C07285=1043.787,311.118,385.391,172.204,41.135,157.884
C07286=1043.780,310.870,385.424,172.200,41.132,157.883
C07287=1043.773,310.622,385.458,172.196,41.130,157.882
C07288=1043.766,310.375,385.491,172.192,41.127,157.881
C07289=1043.759,310.127,385.525,172.189,41.125,157.880
C07290=1043.751,309.879,385.558,172.185,41.122,157.880
C07291=1043.745,309.632,385.591,172.181,41.119,157.879
C07292=1043.738,309.385,385.625,172.177,41.116,157.878
C07293=1043.731,309.136,385.658,172.173,41.113,157.877
C07294=1043.724,308.889,385.691,172.169,41.111,157.876
C07295=1043.717,308.642,385.725,172.165,41.108,157.875
C07296=1043.710,308.393,385.758,172.161,41.106,157.875
C07297=1043.703,308.146,385.792,172.157,41.103,157.874
C07298=1043.696,307.898,385.824,172.153,41.100,157.873
C07299=1043.689,307.651,385.858,172.149,41.098,157.872
C07300=1043.682,307.404,385.892,172.146,41.095,157.872
C07301=1043.675,307.155,385.925,172.142,41.093,157.871
C07302=1043.669,306.908,385.958,172.138,41.090,157.870
C07303=1043.662,306.660,385.991,172.134,41.087,157.869
C07304=1043.654,306.412,386.025,172.130,41.085,157.868
C07305=1043.647,306.165,386.057,172.126,41.082,157.868
C07306=1043.640,305.918,386.091,172.122,41.079,157.867
C07307=1043.632,305.593,386.135,172.117,41.076,157.866
C07308=1043.623,305.268,386.178,172.112,41.073,157.865
C07309=1043.614,304.942,386.222,172.107,41.070,157.864
C07310=1043.605,304.618,386.265,172.102,41.066,157.863
C07311=1043.597,304.370,386.298,172.099,41.063,157.862
C07312=1043.591,304.123,386.331,172.095,41.060,157.861
C07313=1043.584,303.875,386.364,172.091,41.058,157.860
C07314=1043.578,303.627,386.397,172.087,41.056,157.860
C07315=1043.570,303.379,386.431,172.084,41.053,157.859
C07316=1043.564,303.132,386.464,172.080,41.051,157.858
C07317=1043.557,302.885,386.496,172.076,41.048,157.857
C07318=1043.550,302.636,386.529,172.072,41.045,157.856
C07319=1043.544,302.389,386.563,172.068,41.043,157.856
C07320=1043.537,302.141,386.596,172.065,41.040,157.855
C07321=1043.530,301.893,386.628,172.061,41.037,157.854
C07322=1043.523,301.645,386.661,172.057,41.035,157.853
C07323=1043.516,301.398,386.694,172.054,41.032,157.853
C07324=1043.510,301.151,386.727,172.050,41.030,157.852
C07325=1043.503,300.903,386.760,172.046,41.027,157.851
C07326=1043.497,300.655,386.793,172.042,41.025,157.850
C07327=1043.490,300.407,386.826,172.039,41.022,157.850
C07328=1043.483,300.159,386.858,172.035,41.019,157.849
C07329=1043.476,299.912,386.892,172.031,41.017,157.848
C07330=1043.469,299.664,386.925,172.028,41.015,157.847
C07331=1043.463,299.416,386.957,172.024,41.012,157.847
C07332=1043.457,299.169,386.990,172.020,41.009,157.846
C07333=1043.449,298.921,387.023,172.017,41.007,157.845
C07334=1043.443,298.673,387.055,172.013,41.004,157.844
C07335=1043.436,298.426,387.088,172.009,41.001,157.843
C07336=1043.430,298.178,387.121,172.006,40.999,157.843
C07337=1043.423,297.930,387.153,172.002,40.997,157.842
C07338=1043.416,297.683,387.186,171.999,40.994,157.841
C07339=1043.410,297.435,387.219,171.995,40.991,157.840
C07340=1043.403,297.187,387.252,171.991,40.989,157.840
C07341=1043.397,296.939,387.285,171.988,40.987,157.839
C07342=1043.390,296.692,387.317,171.985,40.984,157.838
C07343=1043.383,296.444,387.350,171.981,40.981,157.837
C07344=1043.377,296.197,387.382,171.977,40.979,157.837
C07345=1043.371,295.948,387.415,171.973,40.976,157.836
C07346=1043.364,295.700,387.447,171.970,40.974,157.835
C07347=1043.357,295.453,387.480,171.967,40.971,157.834
C07348=1043.350,295.206,387.512,171.963,40.969,157.834
C07349=1043.343,294.957,387.545,171.959,40.966,157.833
C07350=1043.337,294.709,387.576,171.956,40.964,157.832
C07351=1043.330,294.462,387.609,171.952,40.962,157.832
C07352=1043.323,294.214,387.641,171.949,40.959,157.831
C07353=1043.317,293.966,387.674,171.945,40.957,157.830
C07354=1043.310,293.718,387.706,171.941,40.954,157.829
C07355=1043.303,293.471,387.739,171.938,40.951,157.829
C07356=1043.297,293.223,387.770,171.934,40.949,157.828
C07357=1043.289,292.975,387.803,171.931,40.947,157.827
C07358=1043.283,292.727,387.835,171.927,40.945,157.827
C07359=1043.276,292.479,387.867,171.924,40.942,157.826
C07360=1043.269,292.232,387.899,171.920,40.940,157.825
C07361=1043.263,291.984,387.931,171.916,40.937,157.824
C07362=1043.255,291.736,387.963,171.914,40.935,157.824
C07363=1043.247,291.427,388.003,171.909,40.932,157.823
C07364=1043.239,291.119,388.043,171.905,40.929,157.822
C07365=1043.231,290.810,388.083,171.900,40.926,157.821
C07366=1043.223,290.502,388.123,171.896,40.923,157.820
C07367=1043.215,290.254,388.154,171.892,40.921,157.820
C07368=1043.208,290.006,388.187,171.889,40.918,157.819
C07369=1043.202,289.758,388.219,171.886,40.916,157.818
C07370=1043.196,289.510,388.250,171.882,40.914,157.817
C07371=1043.188,289.263,388.282,171.879,40.911,157.817
C07372=1043.182,289.015,388.314,171.875,40.909,157.816
C07373=1043.176,288.767,388.346,171.871,40.906,157.815
C07374=1043.169,288.520,388.378,171.869,40.904,157.815
C07375=1043.162,288.272,388.409,171.865,40.902,157.814
C07376=1043.155,288.023,388.441,171.861,40.900,157.813
C07377=1043.148,287.775,388.474,171.859,40.897,157.813
C07378=1043.142,287.528,388.505,171.855,40.895,157.812
C07379=1043.135,287.280,388.537,171.851,40.893,157.811
C07380=1043.128,287.032,388.568,171.848,40.890,157.810
C07381=1043.121,286.785,388.600,171.844,40.888,157.810
C07382=1043.114,286.537,388.632,171.841,40.886,157.809
C07383=1043.108,286.289,388.663,171.838,40.883,157.808
C07384=1043.101,286.041,388.695,171.834,40.881,157.808
C07385=1043.094,285.793,388.726,171.831,40.879,157.807
C07386=1043.088,285.545,388.757,171.828,40.877,157.807
C07387=1043.081,285.297,388.789,171.824,40.874,157.806
C07388=1043.074,285.049,388.820,171.820,40.872,157.805
C07389=1043.067,284.802,388.852,171.818,40.870,157.804
C07390=1043.061,284.554,388.884,171.814,40.867,157.804
C07391=1043.054,284.306,388.916,171.811,40.865,157.803
C07392=1043.048,284.058,388.947,171.807,40.863,157.802
C07393=1043.041,283.810,388.979,171.804,40.861,157.802
C07394=1043.034,283.562,389.010,171.801,40.858,157.801
C07395=1043.027,283.314,389.042,171.797,40.856,157.800
C07396=1043.021,283.066,389.073,171.794,40.854,157.800
C07397=1043.014,282.818,389.105,171.791,40.851,157.799
C07398=1043.007,282.570,389.136,171.787,40.849,157.798
C07399=1043.001,282.322,389.167,171.784,40.847,157.798
C07400=1042.994,282.074,389.198,171.781,40.845,157.797
C07401=1042.987,281.826,389.230,171.778,40.842,157.796
C07402=1042.981,281.578,389.261,171.774,40.840,157.796
C07403=1042.974,281.330,389.292,171.770,40.838,157.795
C07404=1042.967,281.082,389.324,171.768,40.836,157.794
C07405=1042.961,280.835,389.355,171.764,40.833,157.794
C07406=1042.954,280.587,389.387,171.761,40.831,157.793
C07407=1042.947,280.338,389.417,171.758,40.829,157.792
C07408=1042.941,280.090,389.449,171.755,40.827,157.792
C07409=1042.935,279.843,389.480,171.751,40.824,157.791
C07410=1042.928,279.595,389.511,171.748,40.822,157.790
C07411=1042.921,279.347,389.543,171.745,40.820,157.790
C07412=1042.915,279.099,389.573,171.742,40.817,157.789
C07413=1042.908,278.851,389.605,171.738,40.815,157.789
C07414=1042.900,278.603,389.636,171.734,40.813,157.788
C07415=1042.894,278.355,389.666,171.732,40.811,157.787
C07416=1042.887,278.107,389.698,171.728,40.808,157.787
C07417=1042.881,277.860,389.729,171.725,40.806,157.786
C07418=1042.874,277.611,389.759,171.722,40.804,157.785
C07419=1042.866,277.314,389.797,171.718,40.802,157.785
C07420=1042.858,277.017,389.834,171.714,40.799,157.784
C07421=1042.850,276.721,389.871,171.710,40.796,157.783
C07422=1042.842,276.424,389.908,171.706,40.793,157.782
C07423=1042.835,276.177,389.938,171.704,40.791,157.782
C07424=1042.829,275.928,389.969,171.700,40.789,157.781
C07425=1042.822,275.680,390.001,171.697,40.787,157.780
C07426=1042.815,275.432,390.032,171.694,40.785,157.780
C07427=1042.808,275.184,390.062,171.691,40.783,157.779
C07428=1042.803,274.936,390.092,171.687,40.781,157.778
C07429=1042.796,274.688,390.124,171.685,40.778,157.778
C07430=1042.789,274.440,390.155,171.681,40.776,157.777
C07431=1042.782,274.192,390.185,171.678,40.774,157.777
C07432=1042.775,273.944,390.216,171.674,40.772,157.776
C07433=1042.769,273.697,390.247,171.672,40.769,157.775
C07434=1042.762,273.448,390.277,171.668,40.767,157.775
C07435=1042.756,273.200,390.308,171.665,40.765,157.774
C07436=1042.749,272.952,390.339,171.662,40.763,157.773
C07437=1042.743,272.705,390.369,171.659,40.761,157.773
C07438=1042.736,272.456,390.400,171.656,40.759,157.772
C07439=1042.729,272.208,390.431,171.653,40.756,157.771
C07440=1042.722,271.960,390.462,171.650,40.754,157.771
C07441=1042.716,271.712,390.492,171.646,40.752,157.770
C07442=1042.709,271.464,390.523,171.644,40.750,157.770
C07443=1042.703,271.216,390.553,171.640,40.748,157.769
C07444=1042.696,270.968,390.583,171.637,40.746,157.768
C07445=1042.690,270.720,390.614,171.635,40.744,157.768
C07446=1042.682,270.472,390.645,171.631,40.741,157.767
C07447=1042.676,270.224,390.675,171.628,40.739,157.767
C07448=1042.669,269.976,390.705,171.625,40.737,157.766
C07449=1042.663,269.728,390.736,171.622,40.735,157.765
C07450=1042.656,269.480,390.766,171.618,40.733,157.765
C07451=1042.650,269.232,390.796,171.616,40.731,157.764
C07452=1042.642,268.984,390.827,171.613,40.728,157.763
C07453=1042.636,268.736,390.858,171.609,40.726,157.763
C07454=1042.629,268.488,390.888,171.607,40.724,157.762
C07455=1042.623,268.240,390.918,171.603,40.723,157.762
C07456=1042.616,267.991,390.949,171.600,40.720,157.761
C07457=1042.610,267.744,390.979,171.598,40.718,157.761
C07458=1042.603,267.495,391.009,171.594,40.716,157.760
C07459=1042.596,267.247,391.040,171.591,40.714,157.759
C07460=1042.590,266.999,391.069,171.588,40.712,157.759
C07461=1042.583,266.751,391.100,171.585,40.710,157.758
C07462=1042.576,266.503,391.130,171.582,40.707,157.757
C07463=1042.565,266.110,391.178,171.577,40.704,157.756
C07464=1042.555,265.716,391.225,171.572,40.701,157.756
C07465=1042.544,265.323,391.273,171.567,40.698,157.755
C07466=1042.534,264.929,391.321,171.563,40.695,157.754
C07467=1042.527,264.681,391.351,171.560,40.692,157.753
C07468=1042.521,264.433,391.381,171.557,40.690,157.752
C07469=1042.514,264.185,391.411,171.554,40.688,157.752
C07470=1042.507,263.937,391.441,171.551,40.686,157.751
C07471=1042.497,263.542,391.489,171.546,40.683,157.750
C07472=1042.486,263.147,391.537,171.542,40.679,157.749
C07473=1042.476,262.752,391.584,171.537,40.676,157.748
C07474=1042.466,262.357,391.633,171.532,40.672,157.747
C07475=1042.459,262.109,391.662,171.529,40.671,157.747
C07476=1042.452,261.861,391.692,171.526,40.669,157.746
C07477=1042.445,261.612,391.722,171.523,40.667,157.746
C07478=1042.439,261.364,391.751,171.520,40.664,157.745
C07479=1042.432,261.116,391.781,171.518,40.663,157.745
C07480=1042.425,260.869,391.811,171.514,40.661,157.744
C07481=1042.418,260.620,391.840,171.511,40.658,157.743
C07482=1042.411,260.371,391.870,171.509,40.657,157.743
C07483=1042.405,260.123,391.899,171.505,40.655,157.742
C07484=1042.398,259.875,391.929,171.502,40.652,157.742
C07485=1042.391,259.627,391.959,171.500,40.651,157.741
C07486=1042.384,259.379,391.989,171.496,40.649,157.741
C07487=1042.377,259.131,392.017,171.494,40.647,157.740
C07488=1042.370,258.883,392.047,171.491,40.644,157.739
C07489=1042.364,258.635,392.076,171.489,40.643,157.739
C07490=1042.357,258.386,392.106,171.485,40.641,157.738
C07491=1042.351,258.138,392.135,171.482,40.638,157.738
C07492=1042.343,257.890,392.166,171.480,40.637,157.737
C07493=1042.337,257.642,392.195,171.476,40.635,157.737
C07494=1042.330,257.394,392.225,171.473,40.632,157.736
C07495=1042.324,257.146,392.254,171.471,40.631,157.736
C07496=1042.317,256.897,392.283,171.468,40.629,157.735
C07497=1042.310,256.649,392.313,171.465,40.627,157.734
C07498=1042.303,256.400,392.342,171.462,40.625,157.734
C07499=1042.297,256.153,392.372,171.459,40.623,157.733
C07500=1042.291,255.905,392.401,171.456,40.621,157.733
C07501=1042.283,255.656,392.430,171.453,40.618,157.732
C07502=1042.276,255.409,392.460,171.451,40.617,157.732
C07503=1042.270,255.160,392.489,171.448,40.615,157.731
C07504=1042.263,254.912,392.518,171.445,40.612,157.730
C07505=1042.257,254.664,392.548,171.442,40.611,157.730
C07506=1042.250,254.415,392.577,171.439,40.609,157.729
C07507=1042.244,254.167,392.606,171.436,40.606,157.729
C07508=1042.237,253.918,392.636,171.434,40.605,157.728
C07509=1042.230,253.671,392.665,171.430,40.603,157.728
C07510=1042.224,253.423,392.695,171.428,40.600,157.727
C07511=1042.217,253.174,392.724,171.425,40.599,157.726
C07512=1042.210,252.926,392.752,171.423,40.597,157.726
C07513=1042.204,252.679,392.782,171.420,40.594,157.725
C07514=1042.197,252.430,392.812,171.416,40.592,157.725
C07515=1042.191,252.182,392.841,171.414,40.591,157.724
C07516=1042.184,251.934,392.870,171.411,40.588,157.724
C07517=1042.177,251.685,392.899,171.408,40.586,157.723
C07518=1042.171,251.437,392.929,171.406,40.585,157.723
C07519=1042.165,251.189,392.958,171.402,40.583,157.722
C07520=1042.158,250.940,392.987,171.400,40.580,157.721
C07521=1042.151,250.692,393.016,171.397,40.579,157.721
C07522=1042.145,250.444,393.045,171.394,40.576,157.720
C07523=1042.138,250.196,393.074,171.392,40.574,157.720
C07524=1042.131,249.947,393.103,171.389,40.572,157.719
C07525=1042.125,249.699,393.132,171.386,40.571,157.719
C07526=1042.119,249.451,393.161,171.383,40.568,157.718
C07527=1042.110,249.157,393.196,171.380,40.566,157.717
C07528=1042.103,248.864,393.231,171.377,40.563,157.717
C07529=1042.095,248.571,393.265,171.374,40.561,157.716
C07530=1042.088,248.276,393.299,171.370,40.558,157.715
C07531=1042.082,248.028,393.328,171.368,40.557,157.715
C07532=1042.075,247.780,393.357,171.365,40.555,157.714
C07533=1042.068,247.532,393.386,171.362,40.552,157.714
C07534=1042.062,247.284,393.415,171.360,40.551,157.713
C07535=1042.056,247.035,393.444,171.357,40.548,157.713
C07536=1042.049,246.787,393.473,171.354,40.546,157.712
C07537=1042.042,246.538,393.502,171.351,40.545,157.711
C07538=1042.036,246.290,393.531,171.348,40.542,157.711
C07539=1042.029,246.043,393.560,171.346,40.540,157.710
C07540=1042.023,245.794,393.589,171.343,40.538,157.710
C07541=1042.017,245.546,393.618,171.341,40.536,157.709
C07542=1042.010,245.298,393.647,171.338,40.534,157.709
C07543=1042.004,245.049,393.676,171.335,40.532,157.708
C07544=1041.997,244.801,393.704,171.333,40.530,157.708
C07545=1041.991,244.553,393.733,171.330,40.528,157.707
C07546=1041.984,244.305,393.762,171.328,40.526,157.706
C07547=1041.977,244.057,393.791,171.325,40.524,157.706
C07548=1041.971,243.807,393.819,171.321,40.522,157.705
C07549=1041.964,243.559,393.848,171.319,40.520,157.705
C07550=1041.958,243.311,393.877,171.316,40.518,157.704
C07551=1041.951,243.064,393.905,171.314,40.516,157.704
C07552=1041.945,242.815,393.934,171.311,40.514,157.703
C07553=1041.938,242.567,393.963,171.308,40.512,157.703
C07554=1041.932,242.319,393.991,171.306,40.511,157.702
C07555=1041.925,242.069,394.020,171.303,40.508,157.701
C07556=1041.918,241.822,394.048,171.301,40.506,157.701
C07557=1041.912,241.573,394.077,171.298,40.504,157.700
C07558=1041.906,241.325,394.106,171.296,40.502,157.700
C07559=1041.899,241.077,394.134,171.293,40.501,157.699
C07560=1041.892,240.829,394.162,171.290,40.498,157.699
C07561=1041.886,240.580,394.191,171.288,40.497,157.698
C07562=1041.878,240.332,394.220,171.285,40.494,157.698
C07563=1041.872,240.083,394.248,171.282,40.492,157.697
C07564=1041.865,239.835,394.276,171.279,40.491,157.697
C07565=1041.859,239.587,394.304,171.276,40.488,157.696
C07566=1041.852,239.339,394.333,171.274,40.487,157.696
C07567=1041.846,239.090,394.361,171.271,40.485,157.695
C07568=1041.839,238.842,394.389,171.269,40.483,157.695
C07569=1041.833,238.594,394.418,171.266,40.481,157.694
C07570=1041.826,238.346,394.446,171.264,40.479,157.693
C07571=1041.819,238.097,394.474,171.261,40.477,157.693
C07572=1041.812,237.849,394.503,171.259,40.475,157.692
C07573=1041.806,237.600,394.531,171.256,40.473,157.692
C07574=1041.799,237.352,394.559,171.253,40.471,157.691
C07575=1041.792,237.104,394.587,171.251,40.469,157.691
C07576=1041.786,236.855,394.615,171.248,40.467,157.690
C07577=1041.779,236.607,394.643,171.246,40.465,157.690
C07578=1041.772,236.359,394.672,171.243,40.464,157.689
C07579=1041.766,236.110,394.700,171.241,40.461,157.689
C07580=1041.759,235.862,394.728,171.238,40.460,157.688
C07581=1041.753,235.614,394.756,171.235,40.458,157.688
C07582=1041.746,235.365,394.784,171.233,40.456,157.687
C07583=1041.738,235.065,394.818,171.230,40.453,157.686
C07584=1041.730,234.766,394.852,171.227,40.451,157.686
C07585=1041.722,234.467,394.886,171.224,40.449,157.685
C07586=1041.714,234.167,394.920,171.220,40.447,157.685
C07587=1041.707,233.919,394.948,171.218,40.444,157.684
C07588=1041.701,233.671,394.976,171.216,40.443,157.684
C07589=1041.695,233.422,395.004,171.214,40.440,157.683
C07590=1041.689,233.174,395.032,171.211,40.439,157.682
C07591=1041.682,232.926,395.060,171.208,40.436,157.682
C07592=1041.675,232.678,395.088,171.206,40.434,157.681
C07593=1041.669,232.429,395.116,171.203,40.433,157.681
C07594=1041.662,232.181,395.144,171.201,40.430,157.680
C07595=1041.656,231.932,395.172,171.198,40.429,157.680
C07596=1041.649,231.684,395.200,171.196,40.426,157.679
C07597=1041.642,231.436,395.228,171.193,40.425,157.679
C07598=1041.635,231.187,395.256,171.190,40.422,157.678
C07599=1041.629,230.939,395.283,171.188,40.421,157.678
C07600=1041.623,230.690,395.312,171.185,40.419,157.677
C07601=1041.616,230.442,395.340,171.183,40.417,157.677
C07602=1041.609,230.193,395.367,171.180,40.415,157.676
C07603=1041.603,229.945,395.395,171.178,40.413,157.676
C07604=1041.596,229.696,395.423,171.175,40.411,157.675
C07605=1041.589,229.448,395.450,171.174,40.409,157.675
C07606=1041.583,229.200,395.478,171.171,40.407,157.674
C07607=1041.577,228.952,395.506,171.168,40.405,157.674
C07608=1041.570,228.703,395.533,171.166,40.403,157.673
C07609=1041.563,228.455,395.561,171.163,40.401,157.672
C07610=1041.557,228.206,395.589,171.161,40.400,157.672
C07611=1041.550,227.958,395.616,171.158,40.397,157.671
C07612=1041.543,227.710,395.644,171.156,40.396,157.671
C07613=1041.536,227.461,395.672,171.153,40.394,157.670
C07614=1041.530,227.213,395.700,171.151,40.392,157.670
C07615=1041.523,226.964,395.727,171.148,40.390,157.669
C07616=1041.516,226.716,395.755,171.147,40.388,157.669
C07617=1041.509,226.467,395.782,171.144,40.386,157.668
C07618=1041.503,226.219,395.809,171.141,40.384,157.668
C07619=1041.497,225.971,395.837,171.139,40.382,157.667
C07620=1041.490,225.722,395.864,171.136,40.380,157.667
C07621=1041.483,225.474,395.892,171.134,40.378,157.666
C07622=1041.476,225.226,395.920,171.131,40.376,157.666
C07623=1041.470,224.977,395.948,171.129,40.375,157.665
C07624=1041.463,224.728,395.975,171.126,40.373,157.665
C07625=1041.456,224.480,396.002,171.125,40.371,157.664
C07626=1041.450,224.232,396.029,171.122,40.369,157.664
C07627=1041.443,223.984,396.057,171.120,40.367,157.663
C07628=1041.437,223.735,396.084,171.117,40.365,157.663
C07629=1041.430,223.486,396.112,171.114,40.363,157.662
C07630=1041.424,223.238,396.139,171.112,40.361,157.662
C07631=1041.417,222.990,396.167,171.109,40.359,157.661
C07632=1041.410,222.741,396.193,171.108,40.357,157.661
C07633=1041.404,222.493,396.221,171.105,40.355,157.660
C07634=1041.397,222.244,396.248,171.103,40.353,157.660
C07635=1041.390,221.996,396.276,171.100,40.352,157.659
C07636=1041.385,221.748,396.303,171.098,40.349,157.659
C07637=1041.378,221.499,396.331,171.095,40.348,157.658
C07638=1041.370,221.251,396.358,171.094,40.345,157.658
C07639=1041.362,220.944,396.392,171.090,40.343,157.657
C07640=1041.354,220.637,396.425,171.087,40.340,157.656
C07641=1041.346,220.330,396.459,171.084,40.338,157.656
C07642=1041.338,220.023,396.493,171.082,40.336,157.655
C07643=1041.332,219.775,396.519,171.079,40.334,157.655
C07644=1041.325,219.526,396.547,171.077,40.332,157.654
C07645=1041.318,219.278,396.574,171.074,40.330,157.654
C07646=1041.312,219.029,396.601,171.072,40.328,157.653
C07647=1041.305,218.780,396.628,171.070,40.326,157.653
C07648=1041.298,218.533,396.655,171.068,40.325,157.652
C07649=1041.292,218.284,396.682,171.065,40.322,157.651
C07650=1041.285,218.035,396.709,171.063,40.321,157.651
C07651=1041.278,217.786,396.736,171.060,40.318,157.650
C07652=1041.271,217.539,396.763,171.059,40.317,157.650
C07653=1041.265,217.290,396.790,171.056,40.315,157.650
C07654=1041.258,217.041,396.816,171.053,40.313,157.649
C07655=1041.251,216.793,396.844,171.051,40.311,157.649
C07656=1041.246,216.544,396.871,171.048,40.309,157.648
C07657=1041.238,216.296,396.898,171.047,40.307,157.648
C07658=1041.232,216.047,396.925,171.044,40.305,157.647
C07659=1041.225,215.800,396.952,171.042,40.303,157.646
C07660=1041.219,215.551,396.979,171.039,40.302,157.646
C07661=1041.211,215.302,397.005,171.038,40.299,157.645
C07662=1041.205,215.054,397.032,171.035,40.298,157.645
C07663=1041.199,214.805,397.059,171.033,40.295,157.644
C07664=1041.192,214.556,397.086,171.030,40.294,157.644
C07665=1041.186,214.309,397.113,171.029,40.292,157.644
C07666=1041.179,214.060,397.140,171.026,40.290,157.643
C07667=1041.172,213.811,397.167,171.024,40.288,157.642
C07668=1041.165,213.563,397.193,171.021,40.286,157.642
C07669=1041.159,213.314,397.220,171.019,40.284,157.641
C07670=1041.152,213.065,397.247,171.017,40.282,157.641
C07671=1041.146,212.818,397.274,171.014,40.280,157.640
C07672=1041.139,212.569,397.301,171.013,40.278,157.640
C07673=1041.132,212.320,397.328,171.010,40.276,157.639
C07674=1041.127,212.072,397.354,171.008,40.274,157.639
C07675=1041.119,211.823,397.382,171.005,40.272,157.638
C07676=1041.113,211.575,397.408,171.004,40.270,157.638
C07677=1041.106,211.326,397.435,171.001,40.268,157.637
C07678=1041.099,211.078,397.461,170.999,40.266,157.637
C07679=1041.093,210.829,397.488,170.997,40.264,157.636
C07680=1041.086,210.581,397.515,170.995,40.262,157.636
C07681=1041.080,210.333,397.541,170.992,40.261,157.635
C07682=1041.073,210.084,397.568,170.989,40.258,157.635
C07683=1041.066,209.835,397.594,170.988,40.257,157.634
C07684=1041.060,209.587,397.621,170.985,40.254,157.634
C07685=1041.053,209.338,397.647,170.983,40.253,157.633
C07686=1041.047,209.090,397.673,170.981,40.250,157.633
C07687=1041.040,208.841,397.700,170.979,40.249,157.632
C07688=1041.033,208.593,397.728,170.976,40.247,157.632
C07689=1041.026,208.345,397.754,170.975,40.245,157.631
C07690=1041.020,208.096,397.781,170.972,40.243,157.631
C07691=1041.013,207.848,397.807,170.970,40.241,157.630
C07692=1041.006,207.599,397.833,170.968,40.239,157.630
C07693=1041.000,207.351,397.859,170.966,40.237,157.629
C07694=1040.993,207.102,397.886,170.963,40.235,157.629
C07695=1040.985,206.800,397.918,170.961,40.233,157.628
C07696=1040.977,206.499,397.949,170.958,40.231,157.628
C07697=1040.969,206.198,397.981,170.955,40.228,157.627
C07698=1040.960,205.896,398.014,170.953,40.226,157.627
C07699=1040.935,204.845,398.120,170.669,40.123,157.593
C07700=1040.929,204.596,398.145,170.667,40.121,157.593
C07701=1040.922,204.348,398.170,170.663,40.120,157.593
C07702=1040.916,204.099,398.196,170.661,40.119,157.592
C07703=1040.910,203.850,398.221,170.657,40.118,157.592
C07704=1040.904,203.602,398.246,170.654,40.117,157.592
C07705=1040.898,203.353,398.271,170.652,40.116,157.591
C07706=1040.892,203.104,398.296,170.648,40.114,157.591
C07707=1040.886,202.856,398.321,170.645,40.113,157.590
C07708=1040.879,202.608,398.346,170.643,40.112,157.590
C07709=1040.873,202.359,398.371,170.639,40.111,157.590
C07710=1040.867,202.110,398.396,170.637,40.110,157.589
C07711=1040.861,201.861,398.421,170.634,40.109,157.589
C07712=1040.855,201.612,398.447,170.630,40.108,157.589
C07713=1040.849,201.364,398.472,170.628,40.106,157.588
C07714=1040.843,201.115,398.496,170.625,40.105,157.588
C07715=1040.837,200.866,398.522,170.621,40.104,157.588
C07716=1040.830,200.617,398.546,170.619,40.103,157.587
C07717=1040.824,200.369,398.571,170.616,40.102,157.587
C07718=1040.817,200.120,398.596,170.613,40.101,157.587
C07719=1040.811,199.871,398.620,170.610,40.099,157.586
C07720=1040.806,199.623,398.645,170.606,40.098,157.586
C07721=1040.799,199.374,398.669,170.604,40.097,157.586
C07722=1040.793,199.125,398.695,170.601,40.096,157.585
C07723=1040.786,198.876,398.719,170.598,40.095,157.585
C07724=1040.780,198.628,398.744,170.595,40.094,157.585
C07725=1040.773,198.379,398.768,170.592,40.093,157.584
C07726=1040.768,198.131,398.793,170.590,40.092,157.584
C07727=1040.762,197.882,398.818,170.586,40.091,157.584
C07728=1040.755,197.633,398.842,170.583,40.090,157.583
C07729=1040.749,197.384,398.867,170.581,40.089,157.583
C07730=1040.742,197.136,398.891,170.577,40.088,157.583
C07731=1040.737,196.887,398.916,170.575,40.087,157.582
C07732=1040.730,196.639,398.941,170.572,40.086,157.582
C07733=1040.724,196.389,398.965,170.568,40.085,157.582
C07734=1040.718,196.141,398.990,170.566,40.084,157.581
C07735=1040.712,195.892,399.014,170.563,40.083,157.581
C07736=1040.706,195.643,399.039,170.560,40.082,157.581
C07737=1040.699,195.395,399.064,170.557,40.081,157.580
C07738=1040.693,195.146,399.088,170.555,40.080,157.580
C07739=1040.686,194.898,399.113,170.551,40.079,157.580
C07740=1040.681,194.648,399.137,170.549,40.078,157.579
C07741=1040.674,194.400,399.161,170.546,40.077,157.579
C07742=1040.668,194.152,399.186,170.542,40.076,157.579
C07743=1040.662,193.903,399.210,170.540,40.075,157.578
C07744=1040.656,193.653,399.235,170.537,40.074,157.578
C07745=1040.650,193.405,399.260,170.534,40.073,157.578
C07746=1040.644,193.156,399.284,170.531,40.072,157.577
C07747=1040.638,192.907,399.309,170.529,40.071,157.577
C07748=1040.632,192.659,399.332,170.526,40.070,157.577
C07749=1040.625,192.410,399.358,170.523,40.069,157.577
C07750=1040.619,192.162,399.381,170.520,40.068,157.576
C07751=1040.613,191.912,399.406,170.518,40.067,157.576
C07752=1040.607,191.664,399.430,170.514,40.066,157.576
C07753=1040.601,191.416,399.455,170.512,40.065,157.575
C07754=1040.595,191.167,399.479,170.509,40.064,157.575
C07755=1040.589,190.917,399.503,170.506,40.063,157.575
C07756=1040.583,190.669,399.527,170.503,40.062,157.574
C07757=1040.577,190.420,399.552,170.501,40.061,157.574
C07758=1040.570,190.172,399.576,170.498,40.060,157.574
C07759=1040.564,189.923,399.601,170.495,40.059,157.573
C07760=1040.557,189.638,399.628,170.492,40.058,157.573
C07761=1040.551,189.354,399.656,170.488,40.057,157.573
C07762=1040.544,189.070,399.683,170.485,40.056,157.572
C07763=1040.537,188.785,399.712,170.482,40.055,157.572
C07764=1040.531,188.537,399.736,170.480,40.054,157.572
C07765=1040.525,188.287,399.760,170.476,40.053,157.571
C07766=1040.519,188.039,399.784,170.474,40.052,157.571
C07767=1040.513,187.790,399.808,170.471,40.051,157.571
C07768=1040.507,187.542,399.832,170.468,40.050,157.570
C07769=1040.500,187.293,399.856,170.465,40.049,157.570
C07770=1040.495,187.044,399.880,170.463,40.048,157.570
C07771=1040.488,186.795,399.904,170.460,40.047,157.569
C07772=1040.483,186.546,399.929,170.457,40.046,157.569
C07773=1040.477,186.297,399.953,170.455,40.045,157.569
C07774=1040.471,186.049,399.977,170.452,40.044,157.569
C07775=1040.465,185.800,400.001,170.449,40.043,157.568
C07776=1040.459,185.551,400.025,170.446,40.042,157.568
C07777=1040.453,185.302,400.049,170.444,40.041,157.568
C07778=1040.447,185.054,400.074,170.441,40.040,157.567
C07779=1040.441,184.805,400.098,170.438,40.039,157.567
C07780=1040.435,184.556,400.122,170.436,40.038,157.567
C07781=1040.429,184.307,400.146,170.432,40.037,157.566
C07782=1040.424,184.059,400.170,170.430,40.037,157.566
C07783=1040.417,183.810,400.194,170.427,40.036,157.566
C07784=1040.412,183.561,400.218,170.425,40.034,157.565
C07785=1040.406,183.313,400.242,170.422,40.033,157.565
C07786=1040.398,183.064,400.265,170.419,40.033,157.565
C07787=1040.392,182.815,400.288,170.417,40.032,157.565
C07788=1040.386,182.566,400.312,170.413,40.031,157.564
C07789=1040.379,182.317,400.336,170.411,40.031,157.564
C07790=1040.373,182.068,400.359,170.408,40.030,157.564
C07791=1040.367,181.819,400.383,170.406,40.029,157.564
C07792=1040.361,181.571,400.406,170.403,40.028,157.563
C07793=1040.354,181.322,400.430,170.400,40.028,157.563
C07794=1040.348,181.073,400.454,170.397,40.027,157.563
C07795=1040.342,180.824,400.477,170.395,40.026,157.563
C07796=1040.336,180.575,400.501,170.392,40.025,157.562
C07797=1040.330,180.327,400.525,170.389,40.024,157.562
C07798=1040.323,180.078,400.547,170.387,40.024,157.562
C07799=1040.317,179.830,400.571,170.384,40.023,157.562
C07800=1040.311,179.580,400.594,170.382,40.022,157.561
C07801=1040.304,179.332,400.618,170.378,40.022,157.561
C07802=1040.298,179.083,400.642,170.376,40.020,157.561
C07803=1040.292,178.834,400.665,170.373,40.020,157.561
C07804=1040.285,178.585,400.689,170.371,40.019,157.560
C07805=1040.280,178.336,400.712,170.368,40.019,157.560
C07806=1040.274,178.088,400.736,170.365,40.018,157.560
C07807=1040.267,177.838,400.759,170.363,40.017,157.560
C07808=1040.261,177.590,400.782,170.360,40.016,157.559
C07809=1040.254,177.340,400.805,170.357,40.016,157.559
C07810=1040.248,177.092,400.829,170.354,40.015,157.559
C07811=1040.243,176.843,400.852,170.352,40.014,157.559
C07812=1040.236,176.594,400.876,170.350,40.013,157.558
C07813=1040.230,176.345,400.899,170.346,40.012,157.558
C07814=1040.224,176.096,400.923,170.344,40.012,157.558
C07815=1040.218,175.848,400.946,170.341,40.011,157.557
C07816=1040.211,175.600,400.969,170.339,40.010,157.557
C07817=1040.205,175.350,400.992,170.336,40.009,157.557
C07818=1040.199,175.102,401.016,170.333,40.009,157.557
C07819=1040.193,174.853,401.039,170.331,40.008,157.556
C07820=1040.187,174.603,401.062,170.329,40.008,157.556
C07821=1040.181,174.355,401.086,170.325,40.007,157.556
C07822=1040.175,174.106,401.109,170.323,40.006,157.556
C07823=1040.168,173.857,401.133,170.320,40.005,157.555
C07824=1040.161,173.573,401.159,170.318,40.004,157.555
C07825=1040.155,173.287,401.185,170.315,40.004,157.555
C07826=1040.147,173.003,401.212,170.311,40.003,157.555
C07827=1040.141,172.718,401.238,170.309,40.002,157.554
C07828=1040.135,172.470,401.262,170.306,40.001,157.554
C07829=1040.127,172.220,401.285,170.303,40.000,157.554
C07830=1040.122,171.971,401.308,170.301,40.000,157.554
C07831=1040.116,171.723,401.331,170.298,39.999,157.553
C07832=1040.110,171.474,401.354,170.296,39.998,157.553
C07833=1040.104,171.225,401.377,170.293,39.997,157.553
C07834=1040.098,170.976,401.400,170.290,39.997,157.553
C07835=1040.091,170.728,401.423,170.288,39.996,157.552
C07836=1040.085,170.479,401.446,170.286,39.995,157.552
C07837=1040.079,170.229,401.470,170.283,39.994,157.552
C07838=1040.073,169.980,401.493,170.280,39.994,157.552
C07839=1040.067,169.732,401.516,170.278,39.993,157.551
C07840=1040.062,169.483,401.539,170.275,39.993,157.551
C07841=1040.055,169.235,401.562,170.273,39.992,157.551
C07842=1040.049,168.985,401.585,170.270,39.991,157.551
C07843=1040.043,168.736,401.608,170.267,39.990,157.550
C07844=1040.037,168.488,401.632,170.265,39.990,157.550
C07845=1040.031,168.239,401.654,170.263,39.989,157.550
C07846=1040.026,167.990,401.677,170.259,39.988,157.550
C07847=1040.018,167.741,401.700,170.257,39.987,157.549
C07848=1040.013,167.492,401.723,170.255,39.987,157.549
C07849=1040.007,167.243,401.746,170.253,39.986,157.549
C07850=1040.001,166.994,401.769,170.250,39.985,157.549
C07851=1039.995,166.746,401.793,170.247,39.984,157.548
C07852=1039.989,166.497,401.815,170.245,39.984,157.548
C07853=1039.983,166.248,401.838,170.242,39.983,157.548
C07854=1039.977,165.999,401.861,170.240,39.982,157.548
C07855=1039.971,165.750,401.884,170.237,39.981,157.547
C07856=1039.965,165.501,401.907,170.235,39.981,157.547
C07857=1039.960,165.252,401.930,170.232,39.980,157.547
C07858=1039.953,165.003,401.952,170.230,39.979,157.547
C07859=1039.947,164.755,401.975,170.228,39.979,157.547
C07860=1039.942,164.506,401.998,170.225,39.978,157.546
C07861=1039.936,164.257,402.021,170.222,39.978,157.546
C07862=1039.929,164.008,402.044,170.220,39.976,157.546
C07863=1039.924,163.759,402.067,170.218,39.976,157.546
C07864=1039.918,163.510,402.090,170.215,39.975,157.545
C07865=1039.912,163.261,402.113,170.212,39.975,157.545
C07866=1039.906,163.012,402.136,170.210,39.974,157.545
C07867=1039.899,162.763,402.158,170.208,39.973,157.545
C07868=1039.894,162.514,402.181,170.205,39.972,157.544
C07869=1039.888,162.265,402.204,170.202,39.972,157.544
C07870=1039.882,162.017,402.227,170.200,39.971,157.544
C07871=1039.876,161.768,402.250,170.198,39.970,157.544
C07872=1039.870,161.519,402.272,170.195,39.969,157.543
C07873=1039.864,161.270,402.295,170.193,39.969,157.543
C07874=1039.859,161.021,402.318,170.190,39.968,157.543
C07875=1039.853,160.772,402.340,170.188,39.967,157.543
C07876=1039.847,160.523,402.363,170.186,39.967,157.542
C07877=1039.841,160.274,402.386,170.183,39.966,157.542
C07878=1039.835,160.025,402.409,170.180,39.965,157.542
C07879=1039.829,159.777,402.431,170.178,39.964,157.542
C07880=1039.823,159.527,402.453,170.176,39.964,157.541
C07881=1039.817,159.279,402.476,170.174,39.963,157.541
C07882=1039.810,159.030,402.498,170.170,39.963,157.541
C07883=1039.805,158.781,402.521,170.168,39.963,157.541
C07884=1039.798,158.532,402.542,170.166,39.961,157.541
C07885=1039.792,158.283,402.565,170.164,39.961,157.540
C07886=1039.786,158.035,402.588,170.161,39.961,157.540
C07887=1039.780,157.785,402.610,170.158,39.960,157.540
C07888=1039.773,157.500,402.635,170.156,39.959,157.540
C07889=1039.765,157.214,402.661,170.153,39.959,157.540
C07890=1039.759,156.930,402.686,170.151,39.958,157.539
C07891=1039.752,156.644,402.712,170.147,39.957,157.539
C07892=1039.746,156.395,402.735,170.145,39.957,157.539
C07893=1039.739,156.147,402.757,170.142,39.956,157.539
C07894=1039.734,155.897,402.779,170.140,39.955,157.538
C07895=1039.727,155.649,402.802,170.138,39.955,157.538
C07896=1039.721,155.399,402.823,170.135,39.955,157.538
C07897=1039.715,155.150,402.846,170.133,39.953,157.538
C07898=1039.709,154.902,402.869,170.130,39.953,157.538
C07899=1039.703,154.653,402.890,170.128,39.953,157.537
C07900=1039.697,154.404,402.913,170.126,39.952,157.537
C07901=1039.691,154.155,402.935,170.124,39.952,157.537
C07902=1039.684,153.906,402.957,170.121,39.951,157.537
C07903=1039.678,153.657,402.979,170.118,39.950,157.537
C07904=1039.673,153.408,403.002,170.116,39.950,157.536
C07905=1039.666,153.159,403.023,170.114,39.949,157.536
C07906=1039.660,152.910,403.046,170.112,39.949,157.536
C07907=1039.654,152.661,403.067,170.108,39.949,157.536
C07908=1039.648,152.412,403.090,170.106,39.948,157.536
C07909=1039.642,152.163,403.112,170.104,39.947,157.535
C07910=1039.636,151.915,403.134,170.102,39.947,157.535
C07911=1039.630,151.666,403.156,170.100,39.946,157.535
C07912=1039.624,151.416,403.177,170.096,39.946,157.535
C07913=1039.618,151.168,403.200,170.094,39.945,157.535
C07914=1039.612,150.918,403.222,170.092,39.944,157.534
C07915=1039.605,150.670,403.244,170.090,39.944,157.534
C07916=1039.599,150.421,403.266,170.088,39.943,157.534
C07917=1039.593,150.171,403.287,170.086,39.943,157.534
C07918=1039.587,149.922,403.310,170.082,39.943,157.534
C07919=1039.581,149.673,403.332,170.080,39.942,157.533
C07920=1039.575,149.424,403.354,170.078,39.941,157.533
C07921=1039.569,149.176,403.376,170.076,39.941,157.533
C07922=1039.563,148.927,403.397,170.074,39.940,157.533
C07923=1039.557,148.678,403.419,170.070,39.940,157.533
C07924=1039.550,148.429,403.441,170.068,39.939,157.532
C07925=1039.545,148.180,403.463,170.066,39.939,157.532
C07926=1039.539,147.930,403.485,170.064,39.939,157.532
C07927=1039.532,147.682,403.507,170.062,39.938,157.532
C07928=1039.526,147.433,403.529,170.059,39.937,157.532
C07929=1039.520,147.184,403.550,170.056,39.937,157.531
C07930=1039.514,146.935,403.572,170.054,39.936,157.531
C07931=1039.508,146.686,403.594,170.052,39.936,157.531
C07932=1039.502,146.437,403.616,170.050,39.935,157.531
C07933=1039.495,146.188,403.638,170.048,39.935,157.531
C07934=1039.489,145.939,403.659,170.046,39.934,157.531
C07935=1039.483,145.690,403.681,170.042,39.934,157.530
C07936=1039.477,145.442,403.703,170.040,39.934,157.530
C07937=1039.471,145.192,403.725,170.038,39.933,157.530
C07938=1039.465,144.943,403.746,170.036,39.933,157.530
C07939=1039.459,144.694,403.768,170.034,39.932,157.530
C07940=1039.452,144.445,403.789,170.032,39.932,157.529
C07941=1039.446,144.196,403.810,170.028,39.931,157.529
C07942=1039.440,143.947,403.832,170.026,39.931,157.529
C07943=1039.434,143.698,403.853,170.024,39.930,157.529
C07944=1039.428,143.450,403.876,170.022,39.930,157.529
C07945=1039.421,143.200,403.897,170.020,39.930,157.529
C07946=1039.415,142.951,403.919,170.018,39.929,157.528
C07947=1039.410,142.703,403.940,170.015,39.929,157.528
C07948=1039.403,142.454,403.962,170.012,39.928,157.528
C07949=1039.397,142.204,403.984,170.010,39.927,157.528
C07950=1039.391,141.955,404.005,170.008,39.927,157.528
C07951=1039.385,141.706,404.027,170.006,39.926,157.527
C07952=1039.378,141.421,404.051,170.003,39.926,157.527
C07953=1039.371,141.135,404.076,170.000,39.926,157.527
C07954=1039.364,140.850,404.101,169.998,39.925,157.527
C07955=1039.357,140.564,404.125,169.995,39.925,157.527
C07956=1039.351,140.315,404.146,169.993,39.924,157.527
C07957=1039.345,140.066,404.168,169.991,39.923,157.526
C07958=1039.339,139.817,404.189,169.988,39.923,157.526
C07959=1039.333,139.567,404.211,169.986,39.922,157.526
C07960=1039.327,139.319,404.232,169.984,39.922,157.526
C07961=1039.321,139.070,404.254,169.981,39.921,157.526
C07962=1039.314,138.821,404.275,169.979,39.921,157.525
C07963=1039.308,138.572,404.296,169.977,39.921,157.525
C07964=1039.302,138.323,404.318,169.974,39.920,157.525
C07965=1039.296,138.074,404.339,169.972,39.920,157.525
C07966=1039.289,137.825,404.360,169.970,39.920,157.525
C07967=1039.284,137.577,404.382,169.968,39.919,157.525
C07968=1039.278,137.327,404.403,169.966,39.919,157.524
C07969=1039.272,137.077,404.424,169.964,39.918,157.524
C07970=1039.265,136.829,404.445,169.961,39.918,157.524
C07971=1039.259,136.580,404.467,169.958,39.918,157.524
C07972=1039.253,136.331,404.488,169.956,39.917,157.524
C07973=1039.246,136.082,404.509,169.954,39.917,157.524
C07974=1039.241,135.833,404.530,169.952,39.916,157.523
C07975=1039.235,135.584,404.551,169.950,39.916,157.523
C07976=1039.228,135.335,404.573,169.948,39.915,157.523
C07977=1039.222,135.086,404.594,169.945,39.915,157.523
C07978=1039.216,134.836,404.615,169.942,39.915,157.523
C07979=1039.209,134.588,404.636,169.940,39.914,157.522
C07980=1039.203,134.338,404.657,169.938,39.914,157.522
C07981=1039.198,134.090,404.679,169.936,39.913,157.522
C07982=1039.191,133.840,404.699,169.934,39.913,157.522
C07983=1039.185,133.591,404.721,169.932,39.913,157.522
C07984=1039.179,133.343,404.742,169.929,39.912,157.522
C07985=1039.172,133.094,404.763,169.927,39.912,157.522
C07986=1039.167,132.845,404.783,169.925,39.912,157.521
C07987=1039.161,132.595,404.805,169.923,39.911,157.521
C07988=1039.154,132.346,404.826,169.921,39.911,157.521
C07989=1039.149,132.097,404.847,169.918,39.910,157.521
C07990=1039.143,131.848,404.868,169.916,39.910,157.521
C07991=1039.136,131.599,404.889,169.913,39.909,157.521
C07992=1039.131,131.350,404.910,169.911,39.909,157.520
C07993=1039.124,131.101,404.932,169.909,39.908,157.520
C07994=1039.118,130.851,404.952,169.907,39.908,157.520
C07995=1039.112,130.603,404.973,169.905,39.908,157.520
C07996=1039.106,130.353,404.993,169.903,39.908,157.520
C07997=1039.099,130.104,405.015,169.901,39.907,157.520
C07998=1039.092,129.856,405.035,169.898,39.907,157.519
C07999=1039.087,129.606,405.056,169.895,39.906,157.519
C08000=1039.080,129.358,405.077,169.893,39.907,157.519
C08001=1039.074,129.108,405.098,169.891,39.906,157.519
C08002=1039.068,128.860,405.119,169.889,39.906,157.519
C08003=1039.062,128.611,405.139,169.887,39.905,157.519
C08004=1039.055,128.362,405.160,169.885,39.905,157.519
C08005=1039.049,128.112,405.181,169.883,39.905,157.518
C08006=1039.043,127.863,405.201,169.880,39.905,157.518
C08007=1039.037,127.614,405.222,169.878,39.904,157.518
C08008=1039.031,127.365,405.242,169.876,39.904,157.518
C08009=1039.024,127.116,405.263,169.873,39.903,157.518
C08010=1039.018,126.866,405.284,169.871,39.903,157.518
C08011=1039.012,126.618,405.305,169.869,39.903,157.518
C08012=1039.005,126.369,405.325,169.867,39.903,157.517
C08013=1039.000,126.120,405.346,169.864,39.902,157.517
C08014=1038.993,125.871,405.367,169.862,39.902,157.517
C08015=1038.986,125.621,405.387,169.860,39.902,157.517
C08016=1038.979,125.336,405.411,169.858,39.901,157.517
C08017=1038.972,125.050,405.434,169.855,39.901,157.517
C08018=1038.965,124.764,405.458,169.853,39.901,157.516
C08019=1038.958,124.478,405.481,169.850,39.900,157.516
C08020=1038.952,124.229,405.503,169.847,39.900,157.516
C08021=1038.946,123.980,405.523,169.845,39.899,157.516
C08022=1038.939,123.731,405.543,169.843,39.899,157.516
C08023=1038.934,123.482,405.565,169.841,39.899,157.516
C08024=1038.927,123.233,405.585,169.839,39.899,157.516
C08025=1038.921,122.984,405.605,169.837,39.898,157.515
C08026=1038.915,122.735,405.626,169.835,39.898,157.515
C08027=1038.909,122.486,405.646,169.832,39.897,157.515
C08028=1038.902,122.236,405.667,169.830,39.897,157.515
C08029=1038.896,121.988,405.687,169.828,39.897,157.515
C08030=1038.890,121.738,405.708,169.826,39.896,157.515
C08031=1038.884,121.490,405.728,169.824,39.896,157.514
C08032=1038.878,121.240,405.749,169.822,39.896,157.514
C08033=1038.872,120.992,405.770,169.820,39.896,157.514
C08034=1038.865,120.742,405.790,169.818,39.895,157.514
C08035=1038.859,120.493,405.810,169.815,39.895,157.514
C08036=1038.853,120.244,405.830,169.813,39.894,157.514
C08037=1038.848,119.995,405.851,169.811,39.894,157.514
C08038=1038.841,119.746,405.872,169.809,39.893,157.513
C08039=1038.835,119.497,405.892,169.807,39.894,157.513
C08040=1038.829,119.248,405.913,169.804,39.893,157.513
C08041=1038.823,118.998,405.933,169.802,39.893,157.513
C08042=1038.817,118.749,405.953,169.800,39.892,157.513
C08043=1038.810,118.501,405.974,169.797,39.892,157.513
C08044=1038.805,118.251,405.995,169.795,39.891,157.512
C08045=1038.799,118.003,406.014,169.793,39.892,157.512
C08046=1038.792,117.753,406.035,169.791,39.891,157.512
C08047=1038.787,117.504,406.055,169.789,39.891,157.512
C08048=1038.780,117.254,406.076,169.787,39.890,157.512
C08049=1038.774,117.006,406.096,169.785,39.890,157.512
C08050=1038.768,116.757,406.116,169.782,39.889,157.512
C08051=1038.762,116.508,406.137,169.780,39.889,157.512
C08052=1038.756,116.259,406.157,169.778,39.889,157.511
C08053=1038.749,116.009,406.178,169.776,39.889,157.511
C08054=1038.743,115.761,406.197,169.774,39.888,157.511
C08055=1038.738,115.511,406.218,169.772,39.888,157.511
C08056=1038.732,115.262,406.238,169.770,39.887,157.511
C08057=1038.726,115.013,406.258,169.767,39.887,157.511
C08058=1038.720,114.764,406.278,169.765,39.887,157.510
C08059=1038.714,114.514,406.299,169.763,39.886,157.510
C08060=1038.708,114.266,406.319,169.761,39.886,157.510
C08061=1038.702,114.017,406.339,169.759,39.886,157.510
C08062=1038.695,113.767,406.359,169.757,39.885,157.510
C08063=1038.690,113.518,406.380,169.755,39.885,157.510
C08064=1038.684,113.269,406.400,169.752,39.884,157.509
C08065=1038.677,113.020,406.420,169.750,39.884,157.509
C08066=1038.671,112.771,406.440,169.748,39.884,157.509
C08067=1038.665,112.522,406.460,169.746,39.883,157.509
C08068=1038.659,112.273,406.481,169.744,39.884,157.509
C08069=1038.653,112.024,406.500,169.742,39.883,157.509
C08070=1038.646,111.774,406.521,169.740,39.883,157.509
C08071=1038.640,111.526,406.541,169.738,39.882,157.508
C08072=1038.634,111.277,406.561,169.736,39.882,157.508
C08073=1038.628,111.027,406.581,169.733,39.882,157.508
C08074=1038.622,110.778,406.601,169.731,39.881,157.508
C08075=1038.616,110.529,406.620,169.729,39.881,157.508
C08076=1038.609,110.279,406.641,169.727,39.881,157.508
C08077=1038.603,110.031,406.660,169.725,39.881,157.508
C08078=1038.597,109.782,406.680,169.723,39.881,157.508
C08079=1038.590,109.533,406.700,169.721,39.880,157.508
C08080=1038.583,109.247,406.723,169.719,39.880,157.507
C08081=1038.576,108.961,406.746,169.715,39.880,157.507
C08082=1038.569,108.675,406.768,169.713,39.880,157.507
C08083=1038.562,108.389,406.791,169.711,39.879,157.507
C08084=1038.555,108.140,406.811,169.709,39.879,157.507
C08085=1038.549,107.890,406.830,169.707,39.879,157.507
C08086=1038.543,107.641,406.850,169.705,39.879,157.507
C08087=1038.536,107.392,406.870,169.703,39.878,157.506
C08088=1038.530,107.143,406.890,169.701,39.878,157.506
C08089=1038.524,106.894,406.909,169.699,39.878,157.506
C08090=1038.518,106.645,406.929,169.696,39.877,157.506
C08091=1038.512,106.396,406.950,169.694,39.878,157.506
C08092=1038.506,106.146,406.969,169.692,39.877,157.506
C08093=1038.499,105.898,406.988,169.690,39.877,157.506
C08094=1038.493,105.648,407.008,169.688,39.876,157.505
C08095=1038.487,105.399,407.028,169.686,39.876,157.505
C08096=1038.481,105.150,407.048,169.684,39.876,157.505
C08097=1038.475,104.901,407.068,169.682,39.875,157.505
C08098=1038.468,104.651,407.087,169.680,39.876,157.505
C08099=1038.462,104.402,407.107,169.677,39.875,157.505
C08100=1038.456,104.154,407.127,169.675,39.875,157.505
C08101=1038.450,103.904,407.146,169.673,39.875,157.505
C08102=1038.444,103.655,407.166,169.671,39.874,157.504
C08103=1038.437,103.406,407.185,169.669,39.874,157.504
C08104=1038.431,103.157,407.205,169.667,39.874,157.504
C08105=1038.425,102.908,407.225,169.665,39.874,157.504
C08106=1038.420,102.659,407.244,169.663,39.873,157.504
C08107=1038.413,102.409,407.264,169.661,39.873,157.504
C08108=1038.406,102.161,407.284,169.658,39.873,157.504
C08109=1038.401,101.911,407.303,169.656,39.872,157.504
C08110=1038.395,101.662,407.323,169.654,39.872,157.503
C08111=1038.389,101.413,407.342,169.652,39.872,157.503
C08112=1038.382,101.163,407.362,169.650,39.872,157.503
C08113=1038.376,100.914,407.381,169.648,39.871,157.503
C08114=1038.370,100.665,407.401,169.646,39.871,157.503
C08115=1038.364,100.416,407.420,169.644,39.871,157.503
C08116=1038.358,100.167,407.440,169.641,39.871,157.503
C08117=1038.351,99.917,407.459,169.639,39.871,157.503
C08118=1038.345,99.669,407.479,169.637,39.870,157.502
C08119=1038.339,99.419,407.498,169.635,39.870,157.502
C08120=1038.333,99.171,407.518,169.633,39.870,157.502
C08121=1038.326,98.921,407.536,169.631,39.869,157.502
C08122=1038.320,98.671,407.556,169.629,39.870,157.502
C08123=1038.313,98.423,407.575,169.627,39.869,157.502
C08124=1038.308,98.173,407.595,169.625,39.869,157.502
C08125=1038.301,97.925,407.614,169.623,39.869,157.502
C08126=1038.295,97.675,407.633,169.620,39.868,157.501
C08127=1038.288,97.426,407.652,169.618,39.869,157.501
C08128=1038.282,97.177,407.672,169.616,39.868,157.501
C08129=1038.277,96.927,407.691,169.614,39.868,157.501
C08130=1038.270,96.678,407.710,169.612,39.868,157.501
C08131=1038.264,96.429,407.730,169.610,39.867,157.501
C08132=1038.258,96.180,407.749,169.608,39.868,157.501
C08133=1038.252,95.931,407.768,169.606,39.867,157.501
C08134=1038.245,95.682,407.788,169.604,39.867,157.501
C08135=1038.239,95.432,407.807,169.602,39.867,157.500
C08136=1038.233,95.183,407.826,169.599,39.866,157.500
C08137=1038.227,94.934,407.846,169.597,39.867,157.500
C08138=1038.220,94.685,407.864,169.595,39.866,157.500
C08139=1038.215,94.436,407.883,169.593,39.866,157.500
C08140=1038.208,94.187,407.903,169.591,39.866,157.500
C08141=1038.202,93.938,407.922,169.589,39.865,157.500
C08142=1038.195,93.688,407.941,169.587,39.866,157.500
C08143=1038.189,93.439,407.960,169.585,39.865,157.499
C08144=1038.183,93.154,407.982,169.583,39.865,157.499
C08145=1038.175,92.867,408.004,169.581,39.865,157.499
C08146=1038.168,92.582,408.026,169.577,39.864,157.499
C08147=1038.161,92.295,408.048,169.575,39.864,157.499
C08148=1038.155,92.046,408.067,169.573,39.864,157.499
C08149=1038.148,91.797,408.087,169.571,39.864,157.499
C08150=1038.143,91.548,408.106,169.569,39.863,157.498
C08151=1038.136,91.299,408.124,169.567,39.863,157.498
C08152=1038.131,91.049,408.144,169.565,39.863,157.498
C08153=1038.124,90.800,408.162,169.563,39.862,157.498
C08154=1038.118,90.551,408.182,169.561,39.863,157.498
C08155=1038.112,90.302,408.201,169.558,39.862,157.498
C08156=1038.106,90.052,408.221,169.556,39.862,157.498
C08157=1038.099,89.803,408.239,169.554,39.862,157.498
C08158=1038.093,89.554,408.258,169.552,39.861,157.497
C08159=1038.086,89.305,408.276,169.550,39.862,157.497
C08160=1038.080,89.056,408.295,169.548,39.861,157.497
C08161=1038.074,88.806,408.314,169.546,39.861,157.497
C08162=1038.068,88.557,408.333,169.544,39.861,157.497
C08163=1038.061,88.308,408.352,169.542,39.861,157.497
C08164=1038.055,88.059,408.370,169.540,39.861,157.497
C08165=1038.049,87.809,408.390,169.537,39.861,157.497
C08166=1038.043,87.560,408.408,169.535,39.860,157.497
C08167=1038.036,87.311,408.427,169.533,39.860,157.497
C08168=1038.030,87.062,408.445,169.531,39.860,157.496
C08169=1038.023,86.813,408.464,169.529,39.860,157.496
C08170=1038.018,86.563,408.483,169.527,39.860,157.496
C08171=1038.011,86.314,408.502,169.525,39.860,157.496
C08172=1038.005,86.065,408.521,169.523,39.859,157.496
C08173=1037.998,85.816,408.539,169.521,39.860,157.496
C08174=1037.992,85.567,408.558,169.520,39.859,157.496
C08175=1037.986,85.318,408.577,169.518,39.859,157.496
C08176=1037.980,85.068,408.596,169.515,39.859,157.496
C08177=1037.974,84.819,408.615,169.513,39.859,157.495
C08178=1037.967,84.570,408.633,169.511,39.858,157.495
C08179=1037.961,84.321,408.652,169.509,39.859,157.495
C08180=1037.955,84.072,408.671,169.507,39.858,157.495
C08181=1037.949,83.823,408.690,169.505,39.858,157.495
C08182=1037.942,83.573,408.708,169.503,39.858,157.495
C08183=1037.936,83.324,408.727,169.501,39.858,157.495
C08184=1037.930,83.075,408.745,169.499,39.858,157.495
C08185=1037.924,82.825,408.764,169.497,39.857,157.494
C08186=1037.917,82.576,408.783,169.495,39.857,157.494
C08187=1037.911,82.327,408.801,169.492,39.857,157.494
C08188=1037.905,82.078,408.820,169.490,39.857,157.494
C08189=1037.898,81.829,408.839,169.488,39.857,157.494
C08190=1037.892,81.580,408.857,169.486,39.857,157.494
C08191=1037.886,81.329,408.876,169.484,39.856,157.494
C08192=1037.880,81.080,408.895,169.482,39.856,157.494
C08193=1037.874,80.831,408.913,169.480,39.856,157.494
C08194=1037.867,80.582,408.932,169.478,39.855,157.493
C08195=1037.861,80.333,408.951,169.476,39.856,157.493
C08196=1037.855,80.085,408.969,169.474,39.855,157.493
C08197=1037.849,79.834,408.987,169.472,39.855,157.493
C08198=1037.843,79.585,409.006,169.469,39.855,157.493
C08199=1037.837,79.336,409.025,169.467,39.855,157.493
C08200=1037.830,79.087,409.043,169.465,39.855,157.493
C08201=1037.824,78.837,409.061,169.463,39.854,157.493
C08202=1037.818,78.588,409.080,169.461,39.854,157.493
C08203=1037.812,78.339,409.099,169.459,39.854,157.492
C08204=1037.806,78.090,409.118,169.457,39.854,157.492
C08205=1037.799,77.840,409.136,169.455,39.854,157.492
C08206=1037.794,77.592,409.154,169.453,39.854,157.492
C08207=1037.787,77.342,409.173,169.452,39.853,157.492
C08208=1037.779,77.056,409.194,169.449,39.853,157.492
C08209=1037.772,76.769,409.215,169.446,39.853,157.492
C08210=1037.765,76.484,409.235,169.444,39.853,157.492
C08211=1037.758,76.198,409.257,169.441,39.853,157.492
C08212=1037.752,75.949,409.276,169.439,39.853,157.492
C08213=1037.745,75.699,409.293,169.437,39.852,157.491
C08214=1037.739,75.451,409.311,169.435,39.853,157.491
C08215=1037.733,75.201,409.329,169.433,39.852,157.491
C08216=1037.726,74.952,409.348,169.431,39.852,157.491
C08217=1037.720,74.703,409.366,169.429,39.852,157.491
C08218=1037.714,74.453,409.384,169.427,39.852,157.491
C08219=1037.707,74.204,409.403,169.425,39.852,157.491
C08220=1037.701,73.954,409.421,169.423,39.852,157.491
C08221=1037.695,73.706,409.439,169.421,39.851,157.491
C08222=1037.689,73.456,409.457,169.419,39.851,157.490
C08223=1037.682,73.207,409.475,169.417,39.851,157.490
C08224=1037.676,72.958,409.493,169.415,39.851,157.490
C08225=1037.670,72.708,409.512,169.413,39.851,157.490
C08226=1037.664,72.459,409.530,169.411,39.851,157.490
C08227=1037.658,72.210,409.548,169.409,39.850,157.490
C08228=1037.651,71.961,409.567,169.407,39.851,157.490
C08229=1037.645,71.711,409.585,169.405,39.850,157.490
C08230=1037.639,71.462,409.602,169.403,39.850,157.490
C08231=1037.633,71.213,409.621,169.401,39.850,157.490
C08232=1037.626,70.964,409.638,169.398,39.850,157.489
C08233=1037.620,70.715,409.657,169.396,39.850,157.489
C08234=1037.614,70.465,409.675,169.394,39.850,157.489
C08235=1037.607,70.216,409.693,169.392,39.850,157.489
C08236=1037.601,69.966,409.711,169.390,39.849,157.489
C08237=1037.595,69.718,409.730,169.388,39.850,157.489
C08238=1037.589,69.468,409.747,169.386,39.849,157.489
C08239=1037.582,69.219,409.766,169.384,39.849,157.489
C08240=1037.576,68.969,409.783,169.382,39.849,157.489
C08241=1037.570,68.720,409.801,169.380,39.849,157.489
C08242=1037.563,68.472,409.819,169.378,39.848,157.488
C08243=1037.557,68.222,409.837,169.375,39.849,157.488
C08244=1037.551,67.972,409.855,169.373,39.849,157.488
C08245=1037.545,67.723,409.874,169.371,39.848,157.488
C08246=1037.538,67.474,409.891,169.369,39.849,157.488
C08247=1037.532,67.224,409.908,169.367,39.848,157.488
C08248=1037.526,66.975,409.927,169.365,39.848,157.488
C08249=1037.520,66.726,409.945,169.363,39.848,157.488
C08250=1037.514,66.477,409.962,169.361,39.848,157.488
C08251=1037.507,66.228,409.981,169.359,39.848,157.487
C08252=1037.501,65.978,409.999,169.357,39.848,157.487
C08253=1037.494,65.729,410.016,169.355,39.848,157.487
C08254=1037.489,65.480,410.034,169.353,39.847,157.487
C08255=1037.481,65.231,410.052,169.351,39.848,157.487
C08256=1037.475,64.981,410.070,169.348,39.847,157.487
C08257=1037.469,64.731,410.087,169.346,39.847,157.487
C08258=1037.463,64.482,410.104,169.344,39.847,157.487
C08259=1037.456,64.233,410.123,169.342,39.847,157.487
C08260=1037.450,63.984,410.141,169.340,39.847,157.487
C08261=1037.444,63.735,410.158,169.338,39.847,157.486
C08262=1037.438,63.485,410.176,169.336,39.847,157.486
C08263=1037.431,63.236,410.193,169.334,39.847,157.486
C08264=1037.425,62.987,410.212,169.332,39.847,157.486
C08265=1037.418,62.737,410.229,169.330,39.847,157.486
C08266=1037.412,62.488,410.246,169.328,39.847,157.486
C08267=1037.405,62.239,410.264,169.326,39.846,157.486
C08268=1037.399,61.989,410.281,169.324,39.847,157.486
C08269=1037.393,61.740,410.299,169.322,39.847,157.486
C08270=1037.386,61.491,410.316,169.320,39.847,157.486
C08271=1037.379,61.241,410.334,169.317,39.847,157.486
C08272=1037.372,60.955,410.354,169.315,39.847,157.486
C08273=1037.365,60.669,410.374,169.312,39.847,157.486
C08274=1037.358,60.383,410.394,169.310,39.846,157.485
C08275=1037.350,60.096,410.414,169.308,39.847,157.485
C08276=1037.343,59.847,410.432,169.306,39.847,157.485
C08277=1037.338,59.598,410.450,169.304,39.846,157.485
C08278=1037.331,59.349,410.467,169.302,39.847,157.485
C08279=1037.324,59.100,410.485,169.299,39.847,157.485
C08280=1037.318,58.850,410.502,169.297,39.846,157.485
C08281=1037.312,58.601,410.519,169.295,39.846,157.485
C08282=1037.305,58.352,410.537,169.293,39.847,157.485
C08283=1037.299,58.103,410.554,169.291,39.846,157.485
C08284=1037.292,57.853,410.572,169.289,39.846,157.485
C08285=1037.285,57.604,410.589,169.287,39.847,157.485
C08286=1037.280,57.355,410.607,169.284,39.846,157.484
C08287=1037.273,57.105,410.624,169.282,39.846,157.484
C08288=1037.267,56.855,410.641,169.280,39.846,157.484
C08289=1037.261,56.606,410.658,169.278,39.846,157.484
C08290=1037.254,56.357,410.675,169.276,39.846,157.484
C08291=1037.249,56.108,410.693,169.274,39.846,157.484
C08292=1037.242,55.858,410.710,169.272,39.846,157.484
C08293=1037.235,55.609,410.728,169.270,39.846,157.484
C08294=1037.229,55.360,410.745,169.268,39.846,157.484
C08295=1037.223,55.110,410.763,169.266,39.846,157.484
C08296=1037.216,54.862,410.780,169.264,39.846,157.484
C08297=1037.210,54.612,410.798,169.262,39.846,157.483
C08298=1037.203,54.362,410.815,169.260,39.846,157.483
C08299=1037.197,54.114,410.832,169.258,39.846,157.483
C08300=1037.191,53.863,410.849,169.256,39.846,157.483
C08301=1037.185,53.615,410.866,169.253,39.845,157.483
C08302=1037.178,53.365,410.883,169.251,39.846,157.483
C08303=1037.172,53.115,410.901,169.249,39.845,157.483
C08304=1037.166,52.867,410.918,169.247,39.845,157.483
C08305=1037.159,52.617,410.936,169.245,39.846,157.483
C08306=1037.153,52.368,410.953,169.243,39.845,157.483
C08307=1037.147,52.118,410.970,169.241,39.845,157.483
C08308=1037.141,51.869,410.987,169.239,39.845,157.483
C08309=1037.134,51.620,411.005,169.237,39.845,157.482
C08310=1037.128,51.371,411.022,169.235,39.845,157.482
C08311=1037.121,51.122,411.039,169.233,39.845,157.482
C08312=1037.116,50.872,411.056,169.231,39.845,157.482
C08313=1037.109,50.622,411.073,169.229,39.845,157.482
C08314=1037.103,50.374,411.090,169.227,39.845,157.482
C08315=1037.097,50.124,411.108,169.224,39.845,157.482
C08316=1037.091,49.875,411.124,169.222,39.845,157.482
C08317=1037.084,49.625,411.142,169.220,39.844,157.482
C08318=1037.079,49.376,411.159,169.218,39.845,157.482
C08319=1037.072,49.127,411.177,169.216,39.844,157.481
C08320=1037.066,48.877,411.193,169.214,39.844,157.481
C08321=1037.060,48.628,411.211,169.212,39.844,157.481
C08322=1037.053,48.379,411.228,169.210,39.844,157.481
C08323=1037.047,48.130,411.245,169.208,39.844,157.481
C08324=1037.041,47.880,411.261,169.206,39.844,157.481
C08325=1037.034,47.630,411.279,169.204,39.844,157.481
C08326=1037.028,47.382,411.296,169.202,39.843,157.481
C08327=1037.022,47.132,411.313,169.200,39.844,157.481
C08328=1037.016,46.883,411.330,169.198,39.844,157.481
C08329=1037.009,46.633,411.348,169.195,39.843,157.480
C08330=1037.003,46.384,411.364,169.193,39.843,157.480
C08331=1036.998,46.135,411.382,169.191,39.843,157.480
C08332=1036.991,45.885,411.399,169.189,39.843,157.480
C08333=1036.985,45.636,411.415,169.187,39.843,157.480
C08334=1036.978,45.387,411.433,169.185,39.843,157.480
C08335=1036.973,45.138,411.450,169.183,39.843,157.480
C08336=1036.963,44.769,411.475,169.180,39.843,157.480
C08337=1036.955,44.401,411.500,169.177,39.842,157.480
C08338=1036.945,44.033,411.525,169.174,39.843,157.479
C08339=1036.935,43.665,411.550,169.170,39.842,157.479
C08340=1036.930,43.415,411.567,169.168,39.842,157.479
C08341=1036.924,43.167,411.584,169.166,39.842,157.479
C08342=1036.917,42.917,411.601,169.164,39.842,157.479
C08343=1036.911,42.668,411.618,169.162,39.842,157.479
C08344=1036.905,42.418,411.634,169.160,39.842,157.479
C08345=1036.898,42.169,411.651,169.158,39.842,157.479
C08346=1036.892,41.920,411.667,169.156,39.842,157.479
C08347=1036.886,41.670,411.685,169.154,39.842,157.479
C08348=1036.880,41.421,411.701,169.152,39.842,157.479
C08349=1036.873,41.172,411.718,169.150,39.842,157.478
C08350=1036.867,40.922,411.735,169.148,39.841,157.478
C08351=1036.861,40.673,411.751,169.146,39.842,157.478
C08352=1036.854,40.423,411.768,169.144,39.842,157.478
C08353=1036.848,40.174,411.784,169.140,39.841,157.478
C08354=1036.841,39.925,411.802,169.138,39.842,157.478
C08355=1036.835,39.675,411.818,169.136,39.842,157.478
C08356=1036.829,39.427,411.835,169.134,39.841,157.478
C08357=1036.822,39.176,411.852,169.132,39.841,157.478
C08358=1036.816,38.927,411.868,169.130,39.842,157.478
C08359=1036.810,38.678,411.885,169.128,39.841,157.478
C08360=1036.804,38.428,411.902,169.126,39.841,157.477
C08361=1036.798,38.179,411.918,169.124,39.842,157.477
C08362=1036.791,37.930,411.935,169.122,39.841,157.477
C08363=1036.785,37.680,411.951,169.120,39.841,157.477
C08364=1036.779,37.431,411.968,169.118,39.841,157.477
C08365=1036.773,37.182,411.985,169.116,39.842,157.477
C08366=1036.766,36.932,412.001,169.114,39.841,157.477
C08367=1036.760,36.683,412.017,169.112,39.841,157.477
C08368=1036.754,36.434,412.034,169.110,39.841,157.477
C08369=1036.747,36.184,412.050,169.108,39.842,157.477
C08370=1036.741,35.935,412.067,169.105,39.841,157.477
C08371=1036.735,35.686,412.083,169.102,39.841,157.477
C08372=1036.728,35.436,412.100,169.100,39.842,157.477
C08373=1036.722,35.187,412.117,169.098,39.842,157.477
C08374=1036.715,34.938,412.132,169.096,39.842,157.476
C08375=1036.709,34.688,412.149,169.094,39.841,157.476
C08376=1036.703,34.438,412.165,169.092,39.842,157.476
C08377=1036.696,34.190,412.182,169.090,39.842,157.476
C08378=1036.690,33.940,412.199,169.088,39.842,157.476
C08379=1036.683,33.691,412.214,169.086,39.841,157.476
C08380=1036.677,33.441,412.231,169.084,39.842,157.476
C08381=1036.671,33.191,412.247,169.082,39.842,157.476
C08382=1036.665,32.942,412.264,169.080,39.842,157.476
C08383=1036.658,32.693,412.280,169.078,39.842,157.476
C08384=1036.652,32.444,412.296,169.075,39.842,157.476
C08385=1036.645,32.194,412.313,169.073,39.842,157.476
C08386=1036.639,31.945,412.329,169.071,39.842,157.476
C08387=1036.633,31.695,412.345,169.069,39.842,157.475
C08388=1036.627,31.446,412.361,169.067,39.842,157.475
C08389=1036.620,31.196,412.378,169.065,39.842,157.475
C08390=1036.614,30.947,412.394,169.063,39.842,157.475
C08391=1036.608,30.698,412.410,169.060,39.842,157.475
C08392=1036.601,30.449,412.426,169.058,39.842,157.475
C08393=1036.595,30.199,412.443,169.056,39.842,157.475
C08394=1036.589,29.950,412.459,169.054,39.842,157.475
C08395=1036.583,29.700,412.476,169.052,39.842,157.475
C08396=1036.574,29.365,412.497,169.049,39.842,157.475
C08397=1036.566,29.029,412.519,169.046,39.842,157.475
C08398=1036.558,28.743,412.538,169.044,39.842,157.474
C08399=1036.552,28.456,412.556,169.041,39.842,157.474
C08400=1036.544,28.169,412.575,169.039,39.842,157.474
C08401=1036.536,27.882,412.594,169.036,39.843,157.474
C08402=1036.530,27.633,412.609,169.034,39.842,157.474
C08403=1036.524,27.383,412.625,169.032,39.842,157.474
C08404=1036.518,27.134,412.641,169.030,39.842,157.474
C08405=1036.511,26.884,412.657,169.028,39.843,157.474
C08406=1036.505,26.635,412.673,169.026,39.843,157.474
C08407=1036.498,26.386,412.689,169.023,39.842,157.474
C08408=1036.492,26.137,412.705,169.021,39.842,157.474
C08409=1036.486,25.888,412.721,169.019,39.843,157.474
C08410=1036.479,25.637,412.738,169.016,39.843,157.474
C08411=1036.473,25.388,412.754,169.014,39.843,157.474
C08412=1036.466,25.139,412.770,169.012,39.843,157.474
C08413=1036.460,24.890,412.786,169.010,39.843,157.473
C08414=1036.454,24.640,412.801,169.008,39.843,157.473
C08415=1036.448,24.391,412.817,169.006,39.843,157.473
C08416=1036.441,24.141,412.833,169.004,39.843,157.473
C08417=1036.435,23.892,412.849,169.002,39.843,157.473
C08418=1036.428,23.643,412.865,168.999,39.844,157.473
C08419=1036.422,23.393,412.881,168.997,39.843,157.473
C08420=1036.416,23.144,412.896,168.995,39.843,157.473
C08421=1036.410,22.894,412.912,168.993,39.844,157.473
C08422=1036.403,22.645,412.928,168.991,39.844,157.473
C08423=1036.397,22.395,412.945,168.989,39.844,157.473
C08424=1036.390,22.146,412.960,168.987,39.843,157.473
C08425=1036.384,21.896,412.976,168.985,39.844,157.473
C08426=1036.378,21.647,412.992,168.982,39.844,157.472
C08427=1036.372,21.398,413.008,168.980,39.844,157.472
C08428=1036.365,21.149,413.023,168.978,39.844,157.472
C08429=1036.359,20.899,413.039,168.975,39.844,157.472
C08430=1036.353,20.650,413.055,168.973,39.844,157.472
C08431=1036.347,20.400,413.071,168.971,39.844,157.472
C08432=1036.339,20.151,413.087,168.969,39.844,157.472
C08433=1036.334,19.901,413.103,168.967,39.844,157.472
C08434=1036.327,19.652,413.118,168.964,39.844,157.472
C08435=1036.321,19.402,413.134,168.962,39.844,157.472
C08436=1036.315,19.153,413.149,168.960,39.844,157.472
C08437=1036.308,18.904,413.165,168.958,39.845,157.472
C08438=1036.302,18.654,413.181,168.956,39.845,157.472
C08439=1036.296,18.405,413.196,168.954,39.845,157.472
C08440=1036.290,18.155,413.212,168.952,39.845,157.472
C08441=1036.283,17.906,413.228,168.949,39.845,157.472
C08442=1036.277,17.657,413.243,168.947,39.845,157.471
C08443=1036.271,17.407,413.259,168.945,39.845,157.471
C08444=1036.264,17.157,413.275,168.943,39.845,157.471
C08445=1036.257,16.908,413.290,168.941,39.845,157.471
C08446=1036.251,16.658,413.307,168.939,39.846,157.471
C08447=1036.245,16.409,413.322,168.937,39.846,157.471
C08448=1036.238,16.160,413.337,168.934,39.846,157.471
C08449=1036.232,15.910,413.353,168.932,39.846,157.471
C08450=1036.226,15.661,413.368,168.930,39.846,157.471
C08451=1036.219,15.411,413.383,168.928,39.846,157.471
C08452=1036.213,15.162,413.400,168.926,39.846,157.471
C08453=1036.207,14.913,413.415,168.923,39.846,157.471
C08454=1036.200,14.663,413.430,168.920,39.846,157.471
C08455=1036.194,14.414,413.446,168.918,39.847,157.471
C08456=1036.188,14.164,413.461,168.916,39.846,157.470
C08457=1036.181,13.915,413.477,168.914,39.846,157.470
C08458=1036.176,13.665,413.493,168.912,39.847,157.470
C08459=1036.169,13.415,413.508,168.910,39.847,157.470
C08460=1036.163,13.166,413.523,168.907,39.847,157.470
C08461=1036.156,12.917,413.538,168.905,39.847,157.470
C08462=1036.149,12.631,413.556,168.903,39.847,157.470
C08463=1036.141,12.346,413.574,168.900,39.848,157.470
C08464=1036.134,12.061,413.591,168.898,39.848,157.470
C08465=1036.126,11.775,413.608,168.895,39.848,157.470
C08466=1036.120,11.526,413.624,168.893,39.848,157.470
C08467=1036.113,11.277,413.639,168.891,39.848,157.470
C08468=1036.107,11.027,413.654,168.889,39.849,157.470
C08469=1036.100,10.778,413.669,168.886,39.849,157.470
C08470=1036.094,10.528,413.684,168.884,39.849,157.470
C08471=1036.088,10.278,413.700,168.882,39.849,157.470
C08472=1036.082,10.029,413.716,168.880,39.849,157.470
C08473=1036.075,9.779,413.730,168.877,39.850,157.470
C08474=1036.069,9.530,413.745,168.875,39.850,157.470
C08475=1036.062,9.281,413.761,168.873,39.850,157.469
C08476=1036.056,9.032,413.776,168.871,39.850,157.469
C08477=1036.050,8.782,413.791,168.869,39.850,157.469
C08478=1036.043,8.533,413.806,168.866,39.851,157.469
C08479=1036.037,8.284,413.821,168.864,39.851,157.469
C08480=1036.030,8.034,413.836,168.862,39.851,157.469
C08481=1036.024,7.784,413.851,168.860,39.851,157.469
C08482=1036.017,7.535,413.867,168.858,39.851,157.469
C08483=1036.011,7.285,413.882,168.855,39.852,157.469
C08484=1036.005,7.036,413.897,168.853,39.852,157.469
C08485=1035.999,6.786,413.912,168.851,39.852,157.469
C08486=1035.992,6.537,413.928,168.849,39.852,157.469
C08487=1035.986,6.287,413.943,168.846,39.852,157.469
C08488=1035.980,6.038,413.957,168.843,39.852,157.469
C08489=1035.974,5.789,413.972,168.841,39.852,157.469
C08490=1035.967,5.539,413.987,168.839,39.852,157.469
C08491=1035.961,5.290,414.003,168.837,39.852,157.469
C08492=1035.954,5.040,414.018,168.834,39.853,157.469
C08493=1035.948,4.791,414.033,168.832,39.853,157.468
C08494=1035.941,4.541,414.048,168.830,39.853,157.468
C08495=1035.935,4.291,414.063,168.828,39.853,157.468
C08496=1035.929,4.042,414.077,168.826,39.853,157.468
C08497=1035.923,3.793,414.093,168.823,39.854,157.468
C08498=1035.916,3.544,414.108,168.821,39.854,157.468
C08499=1035.910,3.294,414.123,168.819,39.854,157.468
C08500=1035.903,3.044,414.138,168.817,39.854,157.468
C08501=1035.897,2.795,414.153,168.815,39.854,157.468
C08502=1035.891,2.546,414.167,168.812,39.855,157.468
C08503=1035.885,2.296,414.182,168.810,39.855,157.468
C08504=1035.879,2.046,414.197,168.808,39.854,157.468
C08505=1035.872,1.797,414.213,168.806,39.854,157.468
C08506=1035.865,1.548,414.228,168.803,39.855,157.468
C08507=1035.860,1.299,414.242,168.801,39.855,157.468
C08508=1035.853,1.049,414.257,168.799,39.855,157.468
C08509=1035.847,0.799,414.272,168.797,39.855,157.468
C08510=1035.841,0.550,414.287,168.795,39.855,157.468
C08511=1035.834,0.300,414.302,168.792,39.856,157.467
C08512=1035.828,0.051,414.317,168.790,39.856,157.467
C08513=1035.822,-0.199,414.332,168.788,39.856,157.467
C08514=1035.816,-0.448,414.347,168.786,39.856,157.467
C08515=1035.810,-0.698,414.362,168.783,39.856,157.467
C08516=1035.804,-0.947,414.377,168.780,39.856,157.467
C08517=1035.798,-1.197,414.392,168.778,39.856,157.467
C08518=1035.791,-1.446,414.407,168.776,39.856,157.467
C08519=1035.785,-1.696,414.422,168.773,39.857,157.467
C08520=1035.779,-1.945,414.436,168.771,39.857,157.467
C08521=1035.773,-2.195,414.451,168.769,39.857,157.467
C08522=1035.766,-2.444,414.466,168.767,39.857,157.467
C08523=1035.761,-2.693,414.481,168.765,39.857,157.467
C08524=1035.754,-2.943,414.496,168.762,39.857,157.467
C08525=1035.748,-3.193,414.511,168.760,39.858,157.467
C08526=1035.741,-3.476,414.527,168.758,39.857,157.466
C08527=1035.734,-3.760,414.543,168.755,39.857,157.466
C08528=1035.727,-4.043,414.560,168.752,39.858,157.466
C08529=1035.719,-4.326,414.577,168.750,39.859,157.466
C08530=1035.713,-4.576,414.591,168.747,39.859,157.466
C08531=1035.706,-4.826,414.605,168.745,39.859,157.466
C08532=1035.700,-5.075,414.620,168.743,39.859,157.466
C08533=1035.694,-5.324,414.635,168.741,39.859,157.466
C08534=1035.687,-5.573,414.649,168.738,39.860,157.466
C08535=1035.681,-5.824,414.663,168.736,39.860,157.466
C08536=1035.675,-6.073,414.678,168.734,39.860,157.466
C08537=1035.668,-6.322,414.692,168.731,39.860,157.466
C08538=1035.661,-6.572,414.707,168.729,39.861,157.466
C08539=1035.655,-6.822,414.722,168.727,39.861,157.466
C08540=1035.649,-7.071,414.735,168.724,39.861,157.466
C08541=1035.642,-7.320,414.750,168.722,39.862,157.466
C08542=1035.636,-7.570,414.765,168.720,39.862,157.466
C08543=1035.630,-7.819,414.779,168.718,39.862,157.466
C08544=1035.624,-8.069,414.794,168.715,39.862,157.466
C08545=1035.617,-8.319,414.809,168.713,39.862,157.466
C08546=1035.611,-8.568,414.822,168.711,39.863,157.466
C08547=1035.605,-8.817,414.837,168.708,39.863,157.466
C08548=1035.598,-9.067,414.852,168.706,39.863,157.466
C08549=1035.592,-9.316,414.865,168.704,39.864,157.466
C08550=1035.586,-9.566,414.880,168.701,39.864,157.466
C08551=1035.578,-9.815,414.894,168.699,39.864,157.465
C08552=1035.573,-10.065,414.908,168.697,39.864,157.465
C08553=1035.567,-10.315,414.923,168.694,39.865,157.465
C08554=1035.560,-10.563,414.937,168.692,39.865,157.465
C08555=1035.554,-10.814,414.951,168.690,39.865,157.465
C08556=1035.548,-11.063,414.966,168.688,39.865,157.465
C08557=1035.541,-11.312,414.980,168.685,39.865,157.465
C08558=1035.535,-11.562,414.994,168.683,39.866,157.465
C08559=1035.529,-11.812,415.009,168.681,39.866,157.465
C08560=1035.522,-12.061,415.023,168.678,39.866,157.465
C08561=1035.516,-12.311,415.038,168.676,39.866,157.465
C08562=1035.510,-12.560,415.051,168.674,39.867,157.465
C08563=1035.503,-12.810,415.066,168.671,39.867,157.465
C08564=1035.498,-13.059,415.080,168.669,39.868,157.465
C08565=1035.491,-13.309,415.094,168.667,39.868,157.465
C08566=1035.484,-13.558,415.109,168.664,39.868,157.465
C08567=1035.479,-13.808,415.123,168.662,39.868,157.465
C08568=1035.472,-14.057,415.137,168.660,39.868,157.465
C08569=1035.466,-14.307,415.151,168.657,39.869,157.465
C08570=1035.459,-14.556,415.165,168.655,39.869,157.465
C08571=1035.454,-14.806,415.179,168.653,39.869,157.465
C08572=1035.447,-15.055,415.194,168.650,39.869,157.465
C08573=1035.441,-15.305,415.208,168.647,39.869,157.464
C08574=1035.435,-15.555,415.222,168.645,39.870,157.464
C08575=1035.429,-15.803,415.236,168.643,39.870,157.464
C08576=1035.422,-16.054,415.250,168.641,39.871,157.464
C08577=1035.415,-16.303,415.264,168.639,39.871,157.464
C08578=1035.409,-16.552,415.278,168.635,39.871,157.464
C08579=1035.403,-16.803,415.292,168.633,39.871,157.464
C08580=1035.397,-17.051,415.306,168.631,39.872,157.464
C08581=1035.390,-17.301,415.319,168.629,39.872,157.464
C08582=1035.384,-17.551,415.333,168.627,39.873,157.464
C08583=1035.377,-17.800,415.348,168.624,39.873,157.464
C08584=1035.372,-18.050,415.362,168.621,39.873,157.464
C08585=1035.365,-18.300,415.375,168.620,39.874,157.464
C08586=1035.358,-18.548,415.389,168.617,39.874,157.464
C08587=1035.352,-18.799,415.403,168.615,39.874,157.464
C08588=1035.346,-19.048,415.417,168.612,39.874,157.464
C08589=1035.339,-19.297,415.431,168.609,39.875,157.464
C08590=1035.332,-19.579,415.446,168.607,39.876,157.464
C08591=1035.325,-19.861,415.462,168.605,39.876,157.464
C08592=1035.318,-20.143,415.477,168.602,39.876,157.464
C08593=1035.311,-20.424,415.493,168.599,39.876,157.464
C08594=1035.305,-20.674,415.507,168.597,39.877,157.464
C08595=1035.298,-20.924,415.521,168.595,39.877,157.464
C08596=1035.292,-21.173,415.535,168.592,39.878,157.464
C08597=1035.286,-21.423,415.549,168.590,39.878,157.464
C08598=1035.280,-21.672,415.562,168.587,39.878,157.464
C08599=1035.273,-21.922,415.576,168.585,39.879,157.464
C08600=1035.267,-22.171,415.590,168.583,39.879,157.464
C08601=1035.260,-22.421,415.604,168.580,39.879,157.464
C08602=1035.254,-22.670,415.617,168.578,39.879,157.464
C08603=1035.248,-22.920,415.631,168.575,39.880,157.464
C08604=1035.242,-23.170,415.645,168.572,39.880,157.463
C08605=1035.235,-23.419,415.658,168.571,39.881,157.464
C08606=1035.229,-23.669,415.673,168.568,39.881,157.463
C08607=1035.223,-23.918,415.686,168.566,39.881,157.463
C08608=1035.217,-24.167,415.700,168.563,39.881,157.463
C08609=1035.211,-24.417,415.714,168.561,39.882,157.463
C08610=1035.204,-24.667,415.727,168.559,39.882,157.463
C08611=1035.198,-24.916,415.740,168.556,39.883,157.463
C08612=1035.192,-25.166,415.755,168.554,39.883,157.463
C08613=1035.185,-25.415,415.769,168.551,39.883,157.463
C08614=1035.179,-25.665,415.782,168.549,39.883,157.463
C08615=1035.173,-25.914,415.796,168.546,39.883,157.463
C08616=1035.167,-26.164,415.809,168.544,39.884,157.463
C08617=1035.160,-26.414,415.823,168.542,39.885,157.463
C08618=1035.155,-26.663,415.837,168.539,39.885,157.463
C08619=1035.148,-26.913,415.850,168.537,39.885,157.463
C08620=1035.142,-27.162,415.864,168.534,39.885,157.463
C08621=1035.135,-27.412,415.877,168.532,39.886,157.463
C08622=1035.129,-27.661,415.890,168.530,39.886,157.463
C08623=1035.122,-27.911,415.904,168.527,39.886,157.463
C08624=1035.116,-28.160,415.917,168.525,39.887,157.463
C08625=1035.111,-28.410,415.931,168.522,39.888,157.463
C08626=1035.104,-28.660,415.945,168.520,39.888,157.463
C08627=1035.098,-28.909,415.958,168.517,39.889,157.463
C08628=1035.091,-29.158,415.971,168.515,39.889,157.463
C08629=1035.085,-29.409,415.984,168.512,39.889,157.463
C08630=1035.079,-29.658,415.997,168.510,39.890,157.463
C08631=1035.073,-29.907,416.011,168.508,39.890,157.463
C08632=1035.066,-30.157,416.024,168.505,39.890,157.463
C08633=1035.060,-30.407,416.038,168.503,39.891,157.463
C08634=1035.053,-30.656,416.051,168.500,39.891,157.463
C08635=1035.046,-30.906,416.065,168.498,39.892,157.463
C08636=1035.040,-31.155,416.078,168.495,39.893,157.463
C08637=1035.034,-31.405,416.090,168.493,39.893,157.463
C08638=1035.028,-31.654,416.104,168.490,39.893,157.463
C08639=1035.021,-31.904,416.117,168.488,39.894,157.463
C08640=1035.015,-32.154,416.131,168.485,39.894,157.463
C08641=1035.009,-32.403,416.144,168.483,39.894,157.463
C08642=1035.002,-32.653,416.157,168.480,39.895,157.463
C08643=1034.996,-32.903,416.170,168.478,39.895,157.463
C08644=1034.990,-33.152,416.183,168.475,39.896,157.463
C08645=1034.984,-33.401,416.197,168.473,39.896,157.463
C08646=1034.978,-33.651,416.210,168.471,39.897,157.463
C08647=1034.971,-33.901,416.224,168.468,39.897,157.463
C08648=1034.966,-34.151,416.237,168.466,39.898,157.463
C08649=1034.959,-34.400,416.250,168.463,39.898,157.463
C08650=1034.953,-34.649,416.263,168.461,39.898,157.463
C08651=1034.946,-34.899,416.277,168.458,39.899,157.463
C08652=1034.940,-35.149,416.289,168.456,39.899,157.463
C08653=1034.934,-35.398,416.303,168.453,39.900,157.462
C08654=1034.927,-35.680,416.317,168.450,39.900,157.462
C08655=1034.920,-35.960,416.332,168.448,39.901,157.462
C08656=1034.913,-36.241,416.347,168.445,39.902,157.463
C08657=1034.905,-36.522,416.362,168.442,39.902,157.462
C08658=1034.900,-36.772,416.374,168.440,39.902,157.462
C08659=1034.893,-37.021,416.388,168.437,39.903,157.462
C08660=1034.887,-37.271,416.401,168.435,39.903,157.462
C08661=1034.881,-37.521,416.414,168.432,39.903,157.462
C08662=1034.875,-37.770,416.427,168.430,39.904,157.462
C08663=1034.869,-38.019,416.440,168.427,39.904,157.462
C08664=1034.862,-38.270,416.453,168.425,39.905,157.462
C08665=1034.856,-38.519,416.466,168.422,39.905,157.462
C08666=1034.850,-38.769,416.479,168.420,39.906,157.462
C08667=1034.844,-39.018,416.492,168.417,39.906,157.462
C08668=1034.838,-39.268,416.505,168.415,39.907,157.462
C08669=1034.832,-39.517,416.518,168.412,39.907,157.462
C08670=1034.825,-39.767,416.530,168.410,39.908,157.462
C08671=1034.818,-40.017,416.544,168.408,39.908,157.462
C08672=1034.812,-40.266,416.557,168.405,39.909,157.462
C08673=1034.806,-40.516,416.569,168.403,39.909,157.462
C08674=1034.799,-40.765,416.582,168.400,39.910,157.462
C08675=1034.793,-41.015,416.595,168.398,39.910,157.462
C08676=1034.787,-41.265,416.607,168.395,39.911,157.462
C08677=1034.781,-41.514,416.620,168.393,39.912,157.462
C08678=1034.775,-41.763,416.632,168.390,39.912,157.462
C08679=1034.768,-42.013,416.646,168.388,39.913,157.462
C08680=1034.762,-42.263,416.659,168.385,39.913,157.462
C08681=1034.756,-42.513,416.672,168.382,39.914,157.462
C08682=1034.749,-42.762,416.684,168.380,39.914,157.462
C08683=1034.743,-43.011,416.697,168.377,39.915,157.462
C08684=1034.737,-43.261,416.710,168.375,39.915,157.462
C08685=1034.731,-43.511,416.722,168.372,39.916,157.462
C08686=1034.724,-43.760,416.735,168.370,39.916,157.462
C08687=1034.718,-44.010,416.747,168.367,39.917,157.462
C08688=1034.712,-44.259,416.761,168.365,39.917,157.462
C08689=1034.705,-44.509,416.773,168.362,39.918,157.462
C08690=1034.699,-44.759,416.785,168.360,39.918,157.462
C08691=1034.693,-45.008,416.798,168.357,39.919,157.462
C08692=1034.687,-45.258,416.811,168.354,39.920,157.462
C08693=1034.681,-45.507,416.823,168.352,39.920,157.462
C08694=1034.674,-45.757,416.836,168.349,39.921,157.462
C08695=1034.668,-46.007,416.849,168.347,39.922,157.462
C08696=1034.662,-46.256,416.861,168.344,39.922,157.462
C08697=1034.656,-46.505,416.874,168.343,39.923,157.462
C08698=1034.650,-46.755,416.887,168.340,39.923,157.462
C08699=1034.644,-47.005,416.899,168.337,39.924,157.462
C08700=1034.637,-47.255,416.911,168.335,39.924,157.462
C08701=1034.631,-47.504,416.924,168.332,39.925,157.462
C08702=1034.625,-47.754,416.937,168.330,39.925,157.462
C08703=1034.618,-48.003,416.949,168.327,39.926,157.462
C08704=1034.612,-48.253,416.961,168.325,39.926,157.462
C08705=1034.606,-48.503,416.975,168.322,39.926,157.462
C08706=1034.600,-48.753,416.987,168.320,39.927,157.462
C08707=1034.594,-49.002,416.999,168.317,39.928,157.462
C08708=1034.588,-49.252,417.012,168.314,39.928,157.462
C08709=1034.582,-49.501,417.025,168.312,39.929,157.462
C08710=1034.575,-49.751,417.037,168.309,39.930,157.462
C08711=1034.569,-50.001,417.050,168.307,39.930,157.462
C08712=1034.563,-50.251,417.062,168.304,39.931,157.462
C08713=1034.556,-50.500,417.074,168.302,39.931,157.462
C08714=1034.551,-50.749,417.086,168.299,39.932,157.462
C08715=1034.544,-50.998,417.099,168.296,39.933,157.462
C08716=1034.538,-51.248,417.111,168.294,39.933,157.462
C08717=1034.532,-51.498,417.123,168.291,39.934,157.462
C08718=1034.525,-51.780,417.137,168.288,39.935,157.462
C08719=1034.517,-52.062,417.150,168.286,39.936,157.462
C08720=1034.510,-52.342,417.164,168.283,39.937,157.462
C08721=1034.503,-52.624,417.178,168.280,39.937,157.462
C08722=1034.496,-52.874,417.190,168.277,39.938,157.462
C08723=1034.490,-53.123,417.202,168.275,39.939,157.462
C08724=1034.484,-53.373,417.215,168.272,39.940,157.463
C08725=1034.477,-53.623,417.226,168.269,39.940,157.462
C08726=1034.471,-53.872,417.238,168.267,39.941,157.463
C08727=1034.465,-54.122,417.251,168.264,39.942,157.463
C08728=1034.459,-54.371,417.263,168.261,39.942,157.463
C08729=1034.452,-54.621,417.275,168.259,39.943,157.463
C08730=1034.446,-54.871,417.287,168.256,39.944,157.463
C08731=1034.439,-55.120,417.299,168.254,39.944,157.463
C08732=1034.433,-55.370,417.311,168.251,39.945,157.463
C08733=1034.427,-55.620,417.324,168.248,39.946,157.463
C08734=1034.420,-55.869,417.336,168.247,39.946,157.463
C08735=1034.414,-56.118,417.347,168.244,39.947,157.463
C08736=1034.408,-56.368,417.360,168.241,39.948,157.463
C08737=1034.402,-56.618,417.371,168.239,39.949,157.463
C08738=1034.395,-56.868,417.383,168.236,39.949,157.463
C08739=1034.389,-57.117,417.395,168.233,39.950,157.463
C08740=1034.383,-57.367,417.407,168.231,39.951,157.463
C08741=1034.377,-57.616,417.419,168.228,39.951,157.463
C08742=1034.370,-57.866,417.431,168.225,39.952,157.463
C08743=1034.364,-58.116,417.443,168.223,39.953,157.463
C08744=1034.358,-58.366,417.455,168.220,39.954,157.463
C08745=1034.351,-58.615,417.467,168.217,39.954,157.463
C08746=1034.345,-58.865,417.479,168.215,39.955,157.463
C08747=1034.339,-59.114,417.491,168.212,39.956,157.463
C08748=1034.332,-59.364,417.503,168.210,39.957,157.463
C08749=1034.326,-59.614,417.514,168.208,39.957,157.463
C08750=1034.320,-59.864,417.527,168.205,39.958,157.463
C08751=1034.314,-60.113,417.538,168.202,39.959,157.463
C08752=1034.308,-60.362,417.550,168.200,39.959,157.463
C08753=1034.302,-60.613,417.562,168.197,39.960,157.463
C08754=1034.295,-60.862,417.574,168.194,39.961,157.463
C08755=1034.289,-61.111,417.586,168.191,39.962,157.463
C08756=1034.283,-61.361,417.598,168.189,39.962,157.463
C08757=1034.277,-61.611,417.609,168.186,39.963,157.463
C08758=1034.270,-61.861,417.621,168.183,39.964,157.463
C08759=1034.264,-62.110,417.633,168.181,39.964,157.463
C08760=1034.258,-62.360,417.644,168.178,39.965,157.463
C08761=1034.252,-62.610,417.657,168.175,39.966,157.463
C08762=1034.246,-62.859,417.668,168.173,39.966,157.463
C08763=1034.239,-63.108,417.680,168.171,39.967,157.463
C08764=1034.233,-63.358,417.691,168.168,39.968,157.464
C08765=1034.228,-63.608,417.704,168.166,39.969,157.464
C08766=1034.221,-63.858,417.715,168.163,39.969,157.464
C08767=1034.215,-64.107,417.727,168.160,39.970,157.464
C08768=1034.209,-64.356,417.738,168.158,39.971,157.464
C08769=1034.203,-64.607,417.750,168.155,39.972,157.464
C08770=1034.196,-64.856,417.762,168.152,39.972,157.464
C08771=1034.190,-65.105,417.774,168.150,39.973,157.464
C08772=1034.184,-65.355,417.785,168.147,39.974,157.464
C08773=1034.178,-65.605,417.798,168.144,39.975,157.464
C08774=1034.172,-65.855,417.809,168.141,39.975,157.464
C08775=1034.166,-66.104,417.820,168.139,39.976,157.464
C08776=1034.159,-66.354,417.832,168.137,39.977,157.464
C08777=1034.154,-66.604,417.844,168.134,39.978,157.464
C08778=1034.147,-66.853,417.856,168.132,39.978,157.464
C08779=1034.142,-67.103,417.867,168.129,39.979,157.464
C08780=1034.135,-67.352,417.879,168.126,39.980,157.464
C08781=1034.129,-67.602,417.890,168.124,39.981,157.464
C08782=1034.122,-67.885,417.903,168.121,39.981,157.464
C08783=1034.115,-68.168,417.916,168.118,39.982,157.464
C08784=1034.109,-68.450,417.929,168.114,39.983,157.464
C08785=1034.102,-68.733,417.942,168.111,39.984,157.464
C08786=1034.096,-68.983,417.955,168.109,39.985,157.464
C08787=1034.090,-69.232,417.965,168.106,39.986,157.464
C08788=1034.083,-69.482,417.977,168.103,39.986,157.464
C08789=1034.078,-69.732,417.988,168.101,39.987,157.464
C08790=1034.071,-69.981,418.000,168.099,39.988,157.464
C08791=1034.065,-70.232,418.012,168.096,39.989,157.464
C08792=1034.059,-70.481,418.024,168.094,39.989,157.464
C08793=1034.053,-70.731,418.035,168.091,39.990,157.464
C08794=1034.047,-70.980,418.046,168.088,39.991,157.464
C08795=1034.041,-71.230,418.058,168.085,39.992,157.464
C08796=1034.036,-71.480,418.069,168.083,39.992,157.464
C08797=1034.029,-71.729,418.081,168.080,39.993,157.464
C08798=1034.023,-71.979,418.092,168.077,39.994,157.464
C08799=1034.017,-72.229,418.103,168.075,39.995,157.465
C08800=1034.011,-72.478,418.115,168.072,39.995,157.464
C08801=1034.006,-72.727,418.126,168.069,39.996,157.464
C08802=1034.000,-72.978,418.138,168.066,39.997,157.465
C08803=1033.994,-73.227,418.149,168.065,39.998,157.465
C08804=1033.987,-73.477,418.160,168.061,39.998,157.465
C08805=1033.981,-73.726,418.171,168.059,39.999,157.465
C08806=1033.975,-73.976,418.183,168.057,40.000,157.465
C08807=1033.970,-74.226,418.195,168.054,40.001,157.465
C08808=1033.963,-74.475,418.205,168.051,40.002,157.465
C08809=1033.957,-74.725,418.216,168.048,40.003,157.465
C08810=1033.951,-74.975,418.227,168.046,40.003,157.465
C08811=1033.945,-75.224,418.239,168.043,40.004,157.465
C08812=1033.938,-75.474,418.250,168.040,40.005,157.465
C08813=1033.933,-75.724,418.261,168.037,40.006,157.465
C08814=1033.926,-75.974,418.272,168.035,40.007,157.465
C08815=1033.920,-76.223,418.283,168.033,40.008,157.465
C08816=1033.914,-76.472,418.295,168.030,40.009,157.465
C08817=1033.908,-76.722,418.306,168.027,40.009,157.465
C08818=1033.902,-76.972,418.317,168.024,40.010,157.465
C08819=1033.895,-77.222,418.328,168.022,40.011,157.465
C08820=1033.890,-77.471,418.339,168.019,40.012,157.465
C08821=1033.883,-77.722,418.350,168.016,40.013,157.465
C08822=1033.877,-77.971,418.361,168.013,40.014,157.465
C08823=1033.872,-78.220,418.372,168.010,40.015,157.465
C08824=1033.865,-78.471,418.383,168.008,40.016,157.465
C08825=1033.859,-78.720,418.394,168.006,40.017,157.466
C08826=1033.853,-78.970,418.406,168.003,40.017,157.466
C08827=1033.847,-79.219,418.417,168.000,40.018,157.466
C08828=1033.841,-79.468,418.427,167.998,40.019,157.466
C08829=1033.834,-79.719,418.438,167.995,40.020,157.466
C08830=1033.829,-79.968,418.449,167.992,40.021,157.466
C08831=1033.823,-80.218,418.460,167.989,40.022,157.466
C08832=1033.817,-80.468,418.471,167.986,40.023,157.466
C08833=1033.810,-80.717,418.481,167.984,40.025,157.466
C08834=1033.804,-80.967,418.493,167.982,40.025,157.466
C08835=1033.797,-81.216,418.503,167.979,40.026,157.466
C08836=1033.792,-81.466,418.513,167.976,40.027,157.466
C08837=1033.786,-81.717,418.524,167.973,40.028,157.466
C08838=1033.779,-81.966,418.535,167.970,40.029,157.466
C08839=1033.773,-82.215,418.545,167.968,40.030,157.466
C08840=1033.767,-82.465,418.557,167.965,40.032,157.467
C08841=1033.760,-82.715,418.567,167.962,40.033,157.467
C08842=1033.755,-82.964,418.578,167.960,40.034,157.467
C08843=1033.748,-83.214,418.589,167.957,40.034,157.467
C08844=1033.742,-83.464,418.599,167.954,40.035,157.467
C08845=1033.737,-83.714,418.609,167.952,40.036,157.467
C08846=1033.729,-83.998,418.623,167.948,40.038,157.467
C08847=1033.722,-84.283,418.634,167.945,40.039,157.467
C08848=1033.715,-84.568,418.647,167.942,40.040,157.467
C08849=1033.708,-84.853,418.659,167.940,40.041,157.467
C08850=1033.702,-85.102,418.669,167.937,40.042,157.467
C08851=1033.696,-85.353,418.679,167.934,40.043,157.467
C08852=1033.689,-85.602,418.690,167.931,40.044,157.467
C08853=1033.683,-85.852,418.701,167.928,40.045,157.467
C08854=1033.678,-86.101,418.712,167.925,40.047,157.468
C08855=1033.671,-86.351,418.722,167.923,40.048,157.468
C08856=1033.665,-86.601,418.732,167.920,40.049,157.468
C08857=1033.659,-86.851,418.743,167.917,40.050,157.468
C08858=1033.653,-87.100,418.753,167.915,40.050,157.468
C08859=1033.647,-87.350,418.765,167.912,40.052,157.468
C08860=1033.640,-87.600,418.774,167.909,40.053,157.468
C08861=1033.635,-87.849,418.785,167.906,40.054,157.468
C08862=1033.628,-88.098,418.795,167.904,40.055,157.468
C08863=1033.622,-88.349,418.806,167.901,40.056,157.468
C08864=1033.616,-88.599,418.817,167.898,40.057,157.468
C08865=1033.610,-88.848,418.827,167.896,40.058,157.468
C08866=1033.604,-89.098,418.837,167.893,40.059,157.468
C08867=1033.598,-89.347,418.848,167.890,40.060,157.468
C08868=1033.592,-89.597,418.859,167.887,40.061,157.468
C08869=1033.586,-89.848,418.869,167.885,40.062,157.469
C08870=1033.580,-90.097,418.879,167.882,40.064,157.469
C08871=1033.574,-90.346,418.890,167.879,40.065,157.469
C08872=1033.568,-90.596,418.900,167.876,40.065,157.469
C08873=1033.562,-90.845,418.911,167.874,40.066,157.469
C08874=1033.556,-91.095,418.920,167.871,40.067,157.469
C08875=1033.550,-91.345,418.931,167.869,40.069,157.469
C08876=1033.544,-91.595,418.942,167.866,40.070,157.469
C08877=1033.538,-91.845,418.952,167.863,40.071,157.469
C08878=1033.532,-92.094,418.963,167.860,40.072,157.469
C08879=1033.526,-92.344,418.972,167.857,40.073,157.469
C08880=1033.520,-92.594,418.983,167.855,40.074,157.469
C08881=1033.514,-92.843,418.993,167.852,40.075,157.469
C08882=1033.508,-93.093,419.004,167.850,40.076,157.470
C08883=1033.501,-93.343,419.014,167.847,40.077,157.470
C08884=1033.496,-93.593,419.024,167.844,40.078,157.470
C08885=1033.490,-93.843,419.035,167.841,40.080,157.470
C08886=1033.484,-94.092,419.045,167.838,40.081,157.470
C08887=1033.478,-94.342,419.055,167.835,40.081,157.470
C08888=1033.472,-94.591,419.065,167.832,40.082,157.470
C08889=1033.466,-94.841,419.075,167.831,40.083,157.470
C08890=1033.460,-95.091,419.086,167.828,40.085,157.470
C08891=1033.454,-95.341,419.096,167.825,40.086,157.470
C08892=1033.448,-95.590,419.106,167.822,40.087,157.470
C08893=1033.443,-95.840,419.116,167.819,40.088,157.470
C08894=1033.436,-96.089,419.127,167.816,40.089,157.470
C08895=1033.431,-96.339,419.137,167.813,40.090,157.471
C08896=1033.424,-96.589,419.146,167.811,40.091,157.471
C08897=1033.419,-96.839,419.157,167.809,40.092,157.471
C08898=1033.413,-97.088,419.167,167.806,40.093,157.471
C08899=1033.407,-97.338,419.178,167.803,40.095,157.471
C08900=1033.401,-97.588,419.187,167.800,40.096,157.471
C08901=1033.395,-97.838,419.197,167.797,40.097,157.471
C08902=1033.389,-98.087,419.208,167.794,40.098,157.471
C08903=1033.383,-98.337,419.217,167.792,40.099,157.471
C08904=1033.377,-98.587,419.227,167.789,40.101,157.471
C08905=1033.371,-98.837,419.237,167.786,40.102,157.471
C08906=1033.364,-99.086,419.247,167.784,40.103,157.471
C08907=1033.358,-99.336,419.257,167.781,40.104,157.472
C08908=1033.353,-99.586,419.267,167.778,40.105,157.472
C08909=1033.347,-99.836,419.277,167.776,40.107,157.472
C08910=1033.339,-100.122,419.289,167.772,40.108,157.472
C08911=1033.332,-100.410,419.300,167.769,40.109,157.472
C08912=1033.326,-100.697,419.311,167.766,40.111,157.472
C08913=1033.318,-100.984,419.322,167.762,40.112,157.472
C08914=1033.312,-101.234,419.332,167.759,40.114,157.472
C08915=1033.307,-101.484,419.342,167.757,40.115,157.472
C08916=1033.301,-101.734,419.352,167.755,40.115,157.472
C08917=1033.294,-101.983,419.362,167.752,40.117,157.473
C08918=1033.288,-102.233,419.372,167.749,40.118,157.473
C08919=1033.283,-102.483,419.382,167.746,40.120,157.473
C08920=1033.276,-102.732,419.391,167.743,40.121,157.473
C08921=1033.270,-102.982,419.401,167.741,40.122,157.473
C08922=1033.265,-103.231,419.410,167.738,40.123,157.473
C08923=1033.259,-103.481,419.420,167.735,40.125,157.473
C08924=1033.253,-103.731,419.431,167.732,40.126,157.473
C08925=1033.247,-103.980,419.440,167.729,40.127,157.473
C08926=1033.240,-104.230,419.450,167.726,40.128,157.473
C08927=1033.234,-104.480,419.459,167.723,40.129,157.474
C08928=1033.229,-104.730,419.469,167.721,40.131,157.474
C08929=1033.223,-104.980,419.479,167.719,40.132,157.474
C08930=1033.217,-105.230,419.489,167.716,40.133,157.474
C08931=1033.211,-105.479,419.498,167.713,40.134,157.474
C08932=1033.205,-105.729,419.507,167.710,40.136,157.474
C08933=1033.199,-105.979,419.518,167.708,40.137,157.474
C08934=1033.193,-106.229,419.527,167.705,40.138,157.474
C08935=1033.187,-106.478,419.537,167.702,40.139,157.474
C08936=1033.181,-106.728,419.546,167.699,40.141,157.475
C08937=1033.175,-106.977,419.555,167.696,40.142,157.475
C08938=1033.169,-107.227,419.565,167.693,40.144,157.475
C08939=1033.164,-107.477,419.575,167.691,40.145,157.475
C08940=1033.157,-107.727,419.585,167.688,40.146,157.475
C08941=1033.151,-107.977,419.594,167.685,40.147,157.475
C08942=1033.145,-108.227,419.604,167.682,40.149,157.475
C08943=1033.140,-108.476,419.613,167.679,40.150,157.475
C08944=1033.133,-108.725,419.623,167.676,40.151,157.475
C08945=1033.128,-108.976,419.631,167.674,40.153,157.476
C08946=1033.121,-109.226,419.641,167.671,40.154,157.476
C08947=1033.115,-109.475,419.651,167.668,40.156,157.476
C08948=1033.109,-109.725,419.660,167.665,40.157,157.476
C08949=1033.103,-109.974,419.669,167.662,40.158,157.476
C08950=1033.097,-110.224,419.679,167.660,40.160,157.476
C08951=1033.091,-110.474,419.688,167.658,40.161,157.476
C08952=1033.085,-110.724,419.697,167.655,40.162,157.476
C08953=1033.080,-110.973,419.707,167.652,40.164,157.476
C08954=1033.073,-111.223,419.716,167.649,40.165,157.477
C08955=1033.067,-111.473,419.726,167.647,40.166,157.477
C08956=1033.061,-111.723,419.735,167.644,40.168,157.477
C08957=1033.056,-111.973,419.744,167.641,40.169,157.477
C08958=1033.050,-112.222,419.753,167.638,40.171,157.477
C08959=1033.044,-112.472,419.763,167.635,40.172,157.477
C08960=1033.037,-112.722,419.772,167.632,40.173,157.477
C08961=1033.032,-112.972,419.781,167.630,40.175,157.477
C08962=1033.026,-113.221,419.790,167.627,40.176,157.477
C08963=1033.020,-113.471,419.800,167.624,40.177,157.478
C08964=1033.014,-113.720,419.809,167.621,40.179,157.478
C08965=1033.008,-113.971,419.818,167.618,40.180,157.478
C08966=1033.002,-114.221,419.828,167.616,40.182,157.478
C08967=1032.997,-114.470,419.837,167.613,40.183,157.478
C08968=1032.991,-114.720,419.846,167.610,40.184,157.478
C08969=1032.985,-114.970,419.855,167.607,40.186,157.478
C08970=1032.978,-115.220,419.865,167.604,40.187,157.478
C08971=1032.973,-115.469,419.873,167.602,40.188,157.479
C08972=1032.966,-115.719,419.882,167.599,40.190,157.479
C08973=1032.960,-115.969,419.892,167.596,40.192,157.479
C08974=1032.954,-116.255,419.902,167.593,40.193,157.479
C08975=1032.948,-116.542,419.913,167.589,40.195,157.479
C08976=1032.940,-116.828,419.923,167.587,40.197,157.479
C08977=1032.933,-117.115,419.934,167.583,40.198,157.479
C08978=1032.928,-117.364,419.942,167.580,40.200,157.480
C08979=1032.922,-117.614,419.952,167.577,40.201,157.480
C08980=1032.915,-117.864,419.960,167.574,40.203,157.480
C08981=1032.910,-118.113,419.969,167.572,40.204,157.480
C08982=1032.904,-118.363,419.979,167.569,40.206,157.480
C08983=1032.898,-118.614,419.988,167.566,40.207,157.480
C08984=1032.892,-118.863,419.997,167.563,40.208,157.480
C08985=1032.886,-119.113,420.006,167.561,40.210,157.480
C08986=1032.880,-119.362,420.014,167.558,40.212,157.481
C08987=1032.874,-119.612,420.023,167.555,40.213,157.481
C08988=1032.868,-119.862,420.033,167.552,40.214,157.481
C08989=1032.863,-120.112,420.041,167.549,40.216,157.481
C08990=1032.857,-120.362,420.050,167.547,40.218,157.481
C08991=1032.850,-120.611,420.059,167.544,40.219,157.481
C08992=1032.845,-120.861,420.067,167.541,40.220,157.481
C08993=1032.839,-121.111,420.077,167.538,40.222,157.482
C08994=1032.833,-121.361,420.086,167.535,40.223,157.482
C08995=1032.827,-121.610,420.094,167.533,40.225,157.482
C08996=1032.821,-121.860,420.103,167.530,40.227,157.482
C08997=1032.815,-122.111,420.112,167.527,40.228,157.482
C08998=1032.810,-122.360,420.121,167.524,40.229,157.482
C08999=1032.803,-122.610,420.129,167.521,40.231,157.482
C09000=1032.797,-122.859,420.138,167.519,40.233,157.482
C09001=1032.792,-123.109,420.147,167.516,40.234,157.483
C09002=1032.786,-123.359,420.156,167.513,40.236,157.483
C09003=1032.780,-123.609,420.165,167.510,40.237,157.483
C09004=1032.774,-123.858,420.173,167.508,40.238,157.483
C09005=1032.768,-124.109,420.182,167.505,40.240,157.483
C09006=1032.763,-124.358,420.191,167.502,40.242,157.483
C09007=1032.756,-124.608,420.200,167.499,40.243,157.483
C09008=1032.751,-124.858,420.208,167.497,40.245,157.484
C09009=1032.745,-125.108,420.217,167.494,40.247,157.484
C09010=1032.739,-125.357,420.226,167.491,40.248,157.484
C09011=1032.733,-125.607,420.234,167.488,40.250,157.484
C09012=1032.727,-125.857,420.243,167.485,40.252,157.484
C09013=1032.721,-126.107,420.251,167.483,40.253,157.484
C09014=1032.715,-126.356,420.260,167.480,40.255,157.485
C09015=1032.709,-126.606,420.268,167.477,40.256,157.485
C09016=1032.703,-126.856,420.277,167.474,40.257,157.485
C09017=1032.698,-127.106,420.286,167.472,40.259,157.485
C09018=1032.691,-127.355,420.295,167.469,40.261,157.485
C09019=1032.686,-127.605,420.303,167.466,40.262,157.485
C09020=1032.680,-127.854,420.311,167.463,40.264,157.485
C09021=1032.675,-128.104,420.321,167.460,40.266,157.486
C09022=1032.671,-128.354,420.330,167.457,40.266,157.485
C09023=1032.667,-128.603,420.340,167.454,40.266,157.485
C09024=1032.662,-128.853,420.351,167.452,40.266,157.485
C09025=1032.660,-129.103,420.362,167.450,40.266,157.485
C09026=1032.658,-129.353,420.375,167.448,40.265,157.485
C09027=1032.657,-129.603,420.386,167.445,40.263,157.484
C09028=1032.656,-129.852,420.400,167.444,40.261,157.484
C09029=1032.656,-130.102,420.413,167.441,40.258,157.484
C09030=1032.657,-130.353,420.428,167.440,40.256,157.483
C09031=1032.659,-130.603,420.442,167.438,40.252,157.482
C09032=1032.660,-130.853,420.458,167.436,40.248,157.482
C09033=1032.663,-131.102,420.474,167.435,40.244,157.481
C09034=1032.666,-131.352,420.491,167.433,40.239,157.480
C09035=1032.671,-131.603,420.508,167.432,40.234,157.479
C09036=1032.675,-131.852,420.525,167.431,40.228,157.478
C09037=1032.681,-132.102,420.544,167.430,40.222,157.477
C09038=1032.354,-132.127,420.253,167.381,40.451,157.513
C09039=1032.348,-131.877,420.234,167.383,40.457,157.514
C09040=1032.344,-131.627,420.216,167.384,40.463,157.515
C09041=1032.340,-131.377,420.199,167.385,40.468,157.516
C09042=1032.337,-131.127,420.182,167.386,40.473,157.517
C09043=1032.333,-130.877,420.166,167.388,40.478,157.518
C09044=1032.331,-130.627,420.151,167.390,40.482,157.519
C09045=1032.330,-130.377,420.136,167.391,40.485,157.519
C09046=1032.330,-130.127,420.121,167.393,40.488,157.520
C09047=1032.330,-129.877,420.108,167.395,40.490,157.520
C09048=1032.331,-129.628,420.095,167.397,40.492,157.521
C09049=1032.331,-129.377,420.082,167.400,40.494,157.521
C09050=1032.334,-129.128,420.070,167.402,40.495,157.521
C09051=1032.336,-128.878,420.059,167.404,40.496,157.522
C09052=1032.339,-128.629,420.048,167.406,40.495,157.522
C09053=1032.343,-128.379,420.038,167.409,40.495,157.522
C09054=1032.348,-128.129,420.029,167.411,40.495,157.522
C09055=1032.353,-127.880,420.019,167.414,40.493,157.522
C09056=1032.359,-127.629,420.010,167.417,40.492,157.522
C09057=1032.364,-127.380,420.002,167.419,40.490,157.521
C09058=1032.371,-127.131,419.993,167.422,40.488,157.521
C09059=1032.376,-126.881,419.985,167.425,40.487,157.521
C09060=1032.382,-126.631,419.977,167.428,40.485,157.521
C09061=1032.388,-126.381,419.968,167.430,40.483,157.521
C09062=1032.395,-126.132,419.959,167.434,40.482,157.521
C09063=1032.400,-125.882,419.951,167.437,40.480,157.520
C09064=1032.406,-125.632,419.942,167.440,40.478,157.520
C09065=1032.412,-125.382,419.934,167.442,40.477,157.520
C09066=1032.418,-125.132,419.925,167.445,40.475,157.520
C09067=1032.423,-124.883,419.916,167.448,40.473,157.520
C09068=1032.430,-124.633,419.908,167.451,40.472,157.520
C09069=1032.435,-124.383,419.899,167.453,40.470,157.520
C09070=1032.441,-124.133,419.890,167.456,40.469,157.520
C09071=1032.447,-123.884,419.882,167.459,40.467,157.519
C09072=1032.453,-123.633,419.873,167.462,40.466,157.519
C09073=1032.458,-123.384,419.864,167.465,40.464,157.519
C09074=1032.465,-123.134,419.855,167.467,40.462,157.519
C09075=1032.471,-122.884,419.847,167.470,40.461,157.519
C09076=1032.477,-122.635,419.837,167.473,40.459,157.519
C09077=1032.482,-122.385,419.829,167.476,40.457,157.518
C09078=1032.488,-122.134,419.820,167.479,40.456,157.518
C09079=1032.494,-121.886,419.811,167.481,40.455,157.518
C09080=1032.500,-121.635,419.803,167.484,40.453,157.518
C09081=1032.505,-121.386,419.794,167.487,40.451,157.518
C09082=1032.511,-121.136,419.784,167.490,40.450,157.518
C09083=1032.517,-120.886,419.777,167.492,40.448,157.518
C09084=1032.524,-120.637,419.767,167.496,40.446,157.517
C09085=1032.529,-120.387,419.759,167.499,40.445,157.517
C09086=1032.535,-120.137,419.749,167.502,40.444,157.517
C09087=1032.541,-119.887,419.740,167.504,40.442,157.517
C09088=1032.547,-119.637,419.732,167.507,40.440,157.517
C09089=1032.553,-119.387,419.723,167.510,40.439,157.517
C09090=1032.558,-119.138,419.714,167.513,40.437,157.517
C09091=1032.565,-118.888,419.705,167.516,40.436,157.517
C09092=1032.570,-118.638,419.696,167.518,40.435,157.516
C09093=1032.577,-118.389,419.687,167.521,40.433,157.516
C09094=1032.583,-118.138,419.678,167.524,40.431,157.516
C09095=1032.588,-117.889,419.669,167.527,40.430,157.516
C09096=1032.594,-117.639,419.660,167.529,40.428,157.516
C09097=1032.600,-117.389,419.651,167.532,40.427,157.516
C09098=1032.606,-117.140,419.642,167.535,40.425,157.516
C09099=1032.613,-116.853,419.632,167.538,40.424,157.516
C09100=1032.620,-116.566,419.621,167.542,40.422,157.515
C09101=1032.626,-116.280,419.610,167.544,40.420,157.515
C09102=1032.633,-115.994,419.600,167.548,40.418,157.515
C09103=1032.639,-115.744,419.591,167.551,40.417,157.515
C09104=1032.645,-115.494,419.582,167.554,40.415,157.515
C09105=1032.651,-115.245,419.573,167.556,40.414,157.515
C09106=1032.657,-114.994,419.564,167.559,40.413,157.515
C09107=1032.663,-114.745,419.554,167.562,40.411,157.514
